LIN {X 0,Y 468.037,Z 394.262,A -85,B 0,C 180,E1 -7685.847,E2 -7685.847} C_VEL
LIN {X 0,Y 468.13,Z 390.567,A -85,B 0,C 180,E1 -7687.99,E2 -7687.99} C_VEL
LIN {X 0,Y 467.913,Z 386.87,A -85,B 0,C 180,E1 -7690.23,E2 -7690.23} C_VEL
LIN {X 0,Y 467.598,Z 384.87,A -85,B 0,C 180,E1 -7691.544,E2 -7691.544} C_VEL
LIN {X 0,Y 467.567,Z 384.871,A -85,B 0,C 180,E1 -7695.053,E2 -7695.053} C_VEL
LIN {X 0,Y 467.59,Z 384.868,A -85,B 0,C 180,E1 -7697.44,E2 -7697.44} C_VEL
LIN {X 0,Y 467.62,Z 384.864,A -85,B 0,C 180,E1 -7700.859,E2 -7700.859} C_VEL
LIN {X 0,Y 467.565,Z 384.872,A -85,B 0,C 180,E1 -7704.26,E2 -7704.26} C_VEL
LIN {X 0,Y 467.583,Z 384.868,A -85,B 0,C 180,E1 -7707.321,E2 -7707.321} C_VEL
LIN {X 0,Y 467.572,Z 384.871,A -85,B 0,C 180,E1 -7710.667,E2 -7710.667} C_VEL
LIN {X 0,Y 467.614,Z 384.861,A -85,B 0,C 180,E1 -7713.2,E2 -7713.2} C_VEL
LIN {X 0,Y 467.591,Z 384.863,A -85,B 0,C 180,E1 -7716.469,E2 -7716.469} C_VEL
LIN {X 0,Y 467.626,Z 384.859,A -85,B 0,C 180,E1 -7719.777,E2 -7719.777} C_VEL
LIN {X 0,Y 467.611,Z 384.862,A -85,B 0,C 180,E1 -7722.507,E2 -7722.507} C_VEL
LIN {X 0,Y 467.612,Z 384.864,A -85,B 0,C 180,E1 -7725.197,E2 -7725.197} C_VEL
LIN {X 0,Y 467.658,Z 384.855,A -85,B 0,C 180,E1 -7727.855,E2 -7727.855} C_VEL
LIN {X 0,Y 467.683,Z 384.852,A -85,B 0,C 180,E1 -7731.357,E2 -7731.357} C_VEL
LIN {X 0,Y 467.745,Z 384.845,A -85,B 0,C 180,E1 -7733.963,E2 -7733.963} C_VEL
LIN {X 0,Y 467.862,Z 384.83,A -85,B 0,C 180,E1 -7737.417,E2 -7737.417} C_VEL
LIN {X 0,Y 467.885,Z 384.831,A -85,B 0,C 180,E1 -7740,E2 -7740} C_VEL
LIN {X 0,Y 467.861,Z 384.829,A -85,B 0,C 180,E1 -7742.583,E2 -7742.583} C_VEL
LIN {X 0,Y 467.746,Z 384.845,A -85,B 0,C 180,E1 -7746.037,E2 -7746.037} C_VEL
LIN {X 0,Y 467.683,Z 384.852,A -85,B 0,C 180,E1 -7748.643,E2 -7748.643} C_VEL
LIN {X 0,Y 467.658,Z 384.855,A -85,B 0,C 180,E1 -7752.145,E2 -7752.145} C_VEL
LIN {X 0,Y 467.658,Z 384.856,A -85,B 0,C 180,E1 -7755.694,E2 -7755.694} C_VEL
LIN {X 0,Y 467.62,Z 384.86,A -85,B 0,C 180,E1 -7758.765,E2 -7758.765} C_VEL
LIN {X 0,Y 467.583,Z 384.868,A -85,B 0,C 180,E1 -7761.269,E2 -7761.269} C_VEL
LIN {X 0,Y 467.576,Z 384.867,A -85,B 0,C 180,E1 -7763.943,E2 -7763.943} C_VEL
LIN {X 0,Y 467.618,Z 384.86,A -85,B 0,C 180,E1 -7766.8,E2 -7766.8} C_VEL
LIN {X 0,Y 467.556,Z 384.868,A -85,B 0,C 180,E1 -7769.738,E2 -7769.738} C_VEL
LIN {X 0,Y 467.585,Z 384.867,A -85,B 0,C 180,E1 -7772.758,E2 -7772.758} C_VEL
LIN {X 0,Y 467.559,Z 384.871,A -85,B 0,C 180,E1 -7775.889,E2 -7775.889} C_VEL
LIN {X 0,Y 467.585,Z 384.867,A -85,B 0,C 180,E1 -7779.145,E2 -7779.145} C_VEL
LIN {X 0,Y 467.588,Z 384.866,A -85,B 0,C 180,E1 -7782.567,E2 -7782.567} C_VEL
LIN {X 0,Y 467.572,Z 384.869,A -85,B 0,C 180,E1 -7785.053,E2 -7785.053} C_VEL
LIN {X 0,Y 467.59,Z 384.867,A -85,B 0,C 180,E1 -7787.44,E2 -7787.44} C_VEL
LIN {X 0,Y 467.569,Z 384.87,A -85,B 0,C 180,E1 -7789.735,E2 -7789.735} C_VEL
LIN {X 0,Y 467.756,Z 387.867,A -85,B 0,C 180,E1 -7791.974,E2 -7791.974} C_VEL
LIN {X 0,Y 467.68,Z 392.609,A -85,B 0,C 180,E1 -7795.177,E2 -7795.177} C_VEL
LIN {X 0,Y 467.509,Z 397.368,A -85,B 0,C 180,E1 -7798.254,E2 -7798.254} C_VEL
LIN {X 0,Y 467.314,Z 402.123,A -85,B 0,C 180,E1 -7801.233,E2 -7801.233} C_VEL
LIN {X 0,Y 467.189,Z 407.463,A -85,B 0,C 180,E1 -7804.501,E2 -7804.501} C_VEL
LIN {X 0,Y 467.08,Z 411.589,A -85,B 0,C 180,E1 -7806.97,E2 -7806.97} C_VEL
LIN {X 0,Y 466.947,Z 416.313,A -85,B 0,C 180,E1 -7809.747,E2 -7809.747} C_VEL
LIN {X 0,Y 466.908,Z 419.366,A -85,B 0,C 180,E1 -7811.43,E2 -7811.43} C_VEL
LIN {X 0,Y 470.476,Z 434.191,A -85,B 0,C 180,E1 -7811.94,E2 -7811.94} C_VEL
LIN {X 0,Y 471.792,Z 441.602,A -85,B 0,C 180,E1 -7812.248,E2 -7812.248} C_VEL
LIN {X 0,Y 471.556,Z 447.954,A -85,B 0,C 180,E1 -7812.5,E2 -7812.5} C_VEL
LIN {X 0,Y 470.818,Z 453.507,A -85,B 0,C 180,E1 -7812.727,E2 -7812.727} C_VEL
LIN {X 0,Y 467.754,Z 462.443,A -85,B 0,C 180,E1 -7813.094,E2 -7813.094} C_VEL
LIN {X 0,Y 464.513,Z 471.086,A -85,B 0,C 180,E1 -7813.54,E2 -7813.54} C_VEL
LIN {X 0,Y 463.507,Z 476.182,A -85,B 0,C 180,E1 -7813.888,E2 -7813.888} C_VEL
LIN {X 0,Y 462.736,Z 487.332,A -85,B 0,C 180,E1 -7814.812,E2 -7814.812} C_VEL
LIN {X 0,Y 462.061,Z 498.248,A -85,B 0,C 180,E1 -7815.915,E2 -7815.915} C_VEL
LIN {X 0,Y 461.458,Z 507.914,A -85,B 0,C 180,E1 -7817.09,E2 -7817.09} C_VEL
LIN {X 0,Y 461.01,Z 516.552,A -85,B 0,C 180,E1 -7818.347,E2 -7818.347} C_VEL
LIN {X 0,Y 460.484,Z 524.187,A -85,B 0,C 180,E1 -7819.669,E2 -7819.669} C_VEL
LIN {X 0,Y 460.097,Z 531.463,A -85,B 0,C 180,E1 -7821.214,E2 -7821.214} C_VEL
LIN {X 0,Y 459.838,Z 537.999,A -85,B 0,C 180,E1 -7822.977,E2 -7822.977} C_VEL
LIN {X 0,Y 459.713,Z 542.902,A -85,B 0,C 180,E1 -7824.737,E2 -7824.737} C_VEL
LIN {X 0,Y 459.585,Z 546.316,A -85,B 0,C 180,E1 -7826.493,E2 -7826.493} C_VEL
LIN {X 0,Y 459.519,Z 548.346,A -85,B 0,C 180,E1 -7828.247,E2 -7828.247} C_VEL
LIN {X 0,Y 459.5,Z 549.045,A -85,B 0,C 180,E1 -7830,E2 -7830} C_VEL
LIN {X 0,Y 459.518,Z 548.421,A -85,B 0,C 180,E1 -7831.753,E2 -7831.753} C_VEL
LIN {X 0,Y 459.585,Z 546.46,A -85,B 0,C 180,E1 -7833.507,E2 -7833.507} C_VEL
LIN {X 0,Y 459.707,Z 543.116,A -85,B 0,C 180,E1 -7835.263,E2 -7835.263} C_VEL
LIN {X 0,Y 459.794,Z 538.292,A -85,B 0,C 180,E1 -7837.024,E2 -7837.024} C_VEL
LIN {X 0,Y 460.086,Z 531.831,A -85,B 0,C 180,E1 -7838.787,E2 -7838.787} C_VEL
LIN {X 0,Y 460.443,Z 524.638,A -85,B 0,C 180,E1 -7840.332,E2 -7840.332} C_VEL
LIN {X 0,Y 461.045,Z 515.741,A -85,B 0,C 180,E1 -7841.876,E2 -7841.876} C_VEL
LIN {X 0,Y 461.588,Z 506.395,A -85,B 0,C 180,E1 -7843.202,E2 -7843.202} C_VEL
LIN {X 0,Y 462.235,Z 496.043,A -85,B 0,C 180,E1 -7844.417,E2 -7844.417} C_VEL
LIN {X 0,Y 462.959,Z 484.619,A -85,B 0,C 180,E1 -7845.519,E2 -7845.519} C_VEL
LIN {X 0,Y 463.727,Z 471.957,A -85,B 0,C 180,E1 -7846.509,E2 -7846.509} C_VEL
LIN {X 0,Y 464.367,Z 459.383,A -85,B 0,C 180,E1 -7847.294,E2 -7847.294} C_VEL
LIN {X 0,Y 464.879,Z 446.27,A -85,B 0,C 180,E1 -7847.929,E2 -7847.929} C_VEL
LIN {X 0,Y 464.878,Z 441.114,A -85,B 0,C 180,E1 -7848.138,E2 -7848.138} C_VEL
LIN {X 0,Y 461.867,Z 427.454,A -85,B 0,C 180,E1 -7848.697,E2 -7848.697} C_VEL
LIN {X 0,Y 459.864,Z 419.255,A -85,B 0,C 180,E1 -7848.975,E2 -7848.975} C_VEL
LIN {X 0,Y 459.964,Z 413.379,A -85,B 0,C 180,E1 -7852.457,E2 -7852.457} C_VEL
LIN {X 0,Y 460.119,Z 408.047,A -85,B 0,C 180,E1 -7855.685,E2 -7855.685} C_VEL
LIN {X 0,Y 460.223,Z 403.902,A -85,B 0,C 180,E1 -7858.255,E2 -7858.255} C_VEL
LIN {X 0,Y 460.45,Z 399.139,A -85,B 0,C 180,E1 -7861.268,E2 -7861.268} C_VEL
LIN {X 0,Y 460.615,Z 394.161,A -85,B 0,C 180,E1 -7864.52,E2 -7864.52} C_VEL
LIN {X 0,Y 460.755,Z 389.63,A -85,B 0,C 180,E1 -7867.599,E2 -7867.599} C_VEL
LIN {X 0,Y 460.574,Z 385.879,A -85,B 0,C 180,E1 -7870.274,E2 -7870.274} C_VEL
LIN {X 0,Y 460.512,Z 385.75,A -85,B 0,C 180,E1 -7873.374,E2 -7873.374} C_VEL
LIN {X 0,Y 460.503,Z 385.751,A -85,B 0,C 180,E1 -7876.625,E2 -7876.625} C_VEL
LIN {X 0,Y 460.544,Z 385.745,A -85,B 0,C 180,E1 -7879.731,E2 -7879.731} C_VEL
LIN {X 0,Y 460.53,Z 385.746,A -85,B 0,C 180,E1 -7882.519,E2 -7882.519} C_VEL
LIN {X 0,Y 460.552,Z 385.742,A -85,B 0,C 180,E1 -7885.624,E2 -7885.624} C_VEL
LIN {X 0,Y 460.54,Z 385.742,A -85,B 0,C 180,E1 -7888.745,E2 -7888.745} C_VEL
LIN {X 0,Y 460.592,Z 385.738,A -85,B 0,C 180,E1 -7892.252,E2 -7892.252} C_VEL
LIN {X 0,Y 460.562,Z 385.74,A -85,B 0,C 180,E1 -7894.705,E2 -7894.705} C_VEL
LIN {X 0,Y 460.514,Z 385.748,A -85,B 0,C 180,E1 -7897.571,E2 -7897.571} C_VEL
LIN {X 0,Y 460.572,Z 385.738,A -85,B 0,C 180,E1 -7900.385,E2 -7900.385} C_VEL
LIN {X 0,Y 460.567,Z 385.738,A -85,B 0,C 180,E1 -7903.146,E2 -7903.146} C_VEL
LIN {X 0,Y 460.561,Z 385.74,A -85,B 0,C 180,E1 -7905.868,E2 -7905.868} C_VEL
LIN {X 0,Y 460.614,Z 385.737,A -85,B 0,C 180,E1 -7908.559,E2 -7908.559} C_VEL
LIN {X 0,Y 460.698,Z 385.725,A -85,B 0,C 180,E1 -7912.109,E2 -7912.109} C_VEL
LIN {X 0,Y 460.7,Z 385.723,A -85,B 0,C 180,E1 -7914.748,E2 -7914.748} C_VEL
LIN {X 0,Y 460.803,Z 385.709,A -85,B 0,C 180,E1 -7917.377,E2 -7917.377} C_VEL
LIN {X 0,Y 460.856,Z 385.708,A -85,B 0,C 180,E1 -7920,E2 -7920} C_VEL
LIN {X 0,Y 460.828,Z 385.706,A -85,B 0,C 180,E1 -7922.622,E2 -7922.622} C_VEL
LIN {X 0,Y 460.713,Z 385.721,A -85,B 0,C 180,E1 -7926.13,E2 -7926.13} C_VEL
LIN {X 0,Y 460.631,Z 385.731,A -85,B 0,C 180,E1 -7928.776,E2 -7928.776} C_VEL
LIN {X 0,Y 460.616,Z 385.733,A -85,B 0,C 180,E1 -7932.445,E2 -7932.445} C_VEL
LIN {X 0,Y 460.603,Z 385.737,A -85,B 0,C 180,E1 -7935.997,E2 -7935.997} C_VEL
LIN {X 0,Y 460.574,Z 385.738,A -85,B 0,C 180,E1 -7938.902,E2 -7938.902} C_VEL
LIN {X 0,Y 460.519,Z 385.746,A -85,B 0,C 180,E1 -7941.485,E2 -7941.485} C_VEL
LIN {X 0,Y 460.545,Z 385.743,A -85,B 0,C 180,E1 -7944.332,E2 -7944.332} C_VEL
LIN {X 0,Y 460.582,Z 385.737,A -85,B 0,C 180,E1 -7947.243,E2 -7947.243} C_VEL
LIN {X 0,Y 460.513,Z 385.744,A -85,B 0,C 180,E1 -7950.24,E2 -7950.24} C_VEL
LIN {X 0,Y 460.532,Z 385.744,A -85,B 0,C 180,E1 -7953.325,E2 -7953.325} C_VEL
LIN {X 0,Y 460.482,Z 385.751,A -85,B 0,C 180,E1 -7956.529,E2 -7956.529} C_VEL
LIN {X 0,Y 460.58,Z 385.739,A -85,B 0,C 180,E1 -7959.857,E2 -7959.857} C_VEL
LIN {X 0,Y 460.514,Z 385.747,A -85,B 0,C 180,E1 -7962.9,E2 -7962.9} C_VEL
LIN {X 0,Y 460.511,Z 385.75,A -85,B 0,C 180,E1 -7965.831,E2 -7965.831} C_VEL
LIN {X 0,Y 460.578,Z 385.905,A -85,B 0,C 180,E1 -7968.391,E2 -7968.391} C_VEL
LIN {X 0,Y 461.077,Z 390.044,A -85,B 0,C 180,E1 -7971.021,E2 -7971.021} C_VEL
LIN {X 0,Y 461.049,Z 394.238,A -85,B 0,C 180,E1 -7973.523,E2 -7973.523} C_VEL
LIN {X 0,Y 460.771,Z 399.769,A -85,B 0,C 180,E1 -7976.695,E2 -7976.695} C_VEL
LIN {X 0,Y 460.523,Z 405.31,A -85,B 0,C 180,E1 -7979.761,E2 -7979.761} C_VEL
LIN {X 0,Y 460.344,Z 410.858,A -85,B 0,C 180,E1 -7982.741,E2 -7982.741} C_VEL
LIN {X 0,Y 460.14,Z 416.417,A -85,B 0,C 180,E1 -7985.645,E2 -7985.645} C_VEL
LIN {X 0,Y 460.006,Z 422.481,A -85,B 0,C 180,E1 -7988.743,E2 -7988.743} C_VEL
LIN {X 0,Y 459.895,Z 427.136,A -85,B 0,C 180,E1 -7991.074,E2 -7991.074} C_VEL
LIN {X 0,Y 463.203,Z 441.778,A -85,B 0,C 180,E1 -7991.567,E2 -7991.567} C_VEL
LIN {X 0,Y 464.921,Z 450.797,A -85,B 0,C 180,E1 -7991.95,E2 -7991.95} C_VEL
LIN {X 0,Y 464.492,Z 463.02,A -85,B 0,C 180,E1 -7992.486,E2 -7992.486} C_VEL
LIN {X 0,Y 463.786,Z 476.719,A -85,B 0,C 180,E1 -7993.267,E2 -7993.267} C_VEL
LIN {X 0,Y 463.109,Z 488.85,A -85,B 0,C 180,E1 -7994.147,E2 -7994.147} C_VEL
LIN {X 0,Y 462.43,Z 499.993,A -85,B 0,C 180,E1 -7995.139,E2 -7995.139} C_VEL
LIN {X 0,Y 461.69,Z 511.188,A -85,B 0,C 180,E1 -7996.352,E2 -7996.352} C_VEL
LIN {X 0,Y 461.077,Z 521.227,A -85,B 0,C 180,E1 -7997.678,E2 -7997.678} C_VEL
LIN {X 0,Y 460.622,Z 529.565,A -85,B 0,C 180,E1 -7999.005,E2 -7999.005} C_VEL
LIN {X 0,Y 460.167,Z 537.534,A -85,B 0,C 180,E1 -8000.55,E2 -8000.55} C_VEL
LIN {X 0,Y 459.848,Z 543.951,A -85,B 0,C 180,E1 -8002.094,E2 -8002.094} C_VEL
LIN {X 0,Y 459.697,Z 549.639,A -85,B 0,C 180,E1 -8003.856,E2 -8003.856} C_VEL
LIN {X 0,Y 459.676,Z 551.888,A -85,B 0,C 180,E1 -8004.737,E2 -8004.737} C_VEL
LIN {X 0,Y 459.548,Z 555.286,A -85,B 0,C 180,E1 -8006.493,E2 -8006.493} C_VEL
LIN {X 0,Y 459.514,Z 557.296,A -85,B 0,C 180,E1 -8008.247,E2 -8008.247} C_VEL
LIN {X 0,Y 459.499,Z 557.962,A -85,B 0,C 180,E1 -8010,E2 -8010} C_VEL
LIN {X 0,Y 459.514,Z 557.297,A -85,B 0,C 180,E1 -8011.753,E2 -8011.753} C_VEL
LIN {X 0,Y 459.548,Z 555.29,A -85,B 0,C 180,E1 -8013.507,E2 -8013.507} C_VEL
LIN {X 0,Y 459.675,Z 551.891,A -85,B 0,C 180,E1 -8015.263,E2 -8015.263} C_VEL
LIN {X 0,Y 459.739,Z 546.998,A -85,B 0,C 180,E1 -8017.025,E2 -8017.025} C_VEL
LIN {X 0,Y 460.042,Z 540.468,A -85,B 0,C 180,E1 -8018.787,E2 -8018.787} C_VEL
LIN {X 0,Y 460.37,Z 533.2,A -85,B 0,C 180,E1 -8020.333,E2 -8020.333} C_VEL
LIN {X 0,Y 460.98,Z 524.2,A -85,B 0,C 180,E1 -8021.877,E2 -8021.877} C_VEL
LIN {X 0,Y 461.502,Z 514.753,A -85,B 0,C 180,E1 -8023.204,E2 -8023.204} C_VEL
LIN {X 0,Y 462.124,Z 504.293,A -85,B 0,C 180,E1 -8024.42,E2 -8024.42} C_VEL
LIN {X 0,Y 462.87,Z 492.752,A -85,B 0,C 180,E1 -8025.522,E2 -8025.522} C_VEL
LIN {X 0,Y 463.62,Z 479.947,A -85,B 0,C 180,E1 -8026.513,E2 -8026.513} C_VEL
LIN {X 0,Y 464.325,Z 466.553,A -85,B 0,C 180,E1 -8027.331,E2 -8027.331} C_VEL
LIN {X 0,Y 464.838,Z 453.547,A -85,B 0,C 180,E1 -8027.941,E2 -8027.941} C_VEL
LIN {X 0,Y 464.782,Z 449.968,A -85,B 0,C 180,E1 -8028.085,E2 -8028.085} C_VEL
LIN {X 0,Y 461.942,Z 435.895,A -85,B 0,C 180,E1 -8028.648,E2 -8028.648} C_VEL
LIN {X 0,Y 459.916,Z 427.098,A -85,B 0,C 180,E1 -8028.94,E2 -8028.94} C_VEL
LIN {X 0,Y 460.047,Z 420.117,A -85,B 0,C 180,E1 -8032.452,E2 -8032.452} C_VEL
LIN {X 0,Y 460.23,Z 413.791,A -85,B 0,C 180,E1 -8035.714,E2 -8035.714} C_VEL
LIN {X 0,Y 460.374,Z 408.996,A -85,B 0,C 180,E1 -8038.245,E2 -8038.245} C_VEL
LIN {X 0,Y 460.633,Z 403.347,A -85,B 0,C 180,E1 -8041.306,E2 -8041.306} C_VEL
LIN {X 0,Y 460.892,Z 397.528,A -85,B 0,C 180,E1 -8044.57,E2 -8044.57} C_VEL
LIN {X 0,Y 461.125,Z 392.357,A -85,B 0,C 180,E1 -8047.577,E2 -8047.577} C_VEL
LIN {X 0,Y 460.973,Z 388.68,A -85,B 0,C 180,E1 -8049.817,E2 -8049.817} C_VEL
LIN {X 0,Y 460.57,Z 385.745,A -85,B 0,C 180,E1 -8051.733,E2 -8051.733} C_VEL
LIN {X 0,Y 460.514,Z 385.748,A -85,B 0,C 180,E1 -8055.411,E2 -8055.411} C_VEL
LIN {X 0,Y 460.536,Z 385.745,A -85,B 0,C 180,E1 -8058.397,E2 -8058.397} C_VEL
LIN {X 0,Y 460.549,Z 385.745,A -85,B 0,C 180,E1 -8061.269,E2 -8061.269} C_VEL
LIN {X 0,Y 460.515,Z 385.749,A -85,B 0,C 180,E1 -8064.555,E2 -8064.555} C_VEL
LIN {X 0,Y 460.533,Z 385.747,A -85,B 0,C 180,E1 -8067.716,E2 -8067.716} C_VEL
LIN {X 0,Y 460.541,Z 385.747,A -85,B 0,C 180,E1 -8070.769,E2 -8070.769} C_VEL
LIN {X 0,Y 460.557,Z 385.742,A -85,B 0,C 180,E1 -8073.734,E2 -8073.734} C_VEL
LIN {X 0,Y 460.545,Z 385.741,A -85,B 0,C 180,E1 -8076.624,E2 -8076.624} C_VEL
LIN {X 0,Y 460.554,Z 385.741,A -85,B 0,C 180,E1 -8079.453,E2 -8079.453} C_VEL
LIN {X 0,Y 460.561,Z 385.742,A -85,B 0,C 180,E1 -8082.23,E2 -8082.23} C_VEL
LIN {X 0,Y 460.574,Z 385.738,A -85,B 0,C 180,E1 -8084.965,E2 -8084.965} C_VEL
LIN {X 0,Y 460.613,Z 385.736,A -85,B 0,C 180,E1 -8088.559,E2 -8088.559} C_VEL
LIN {X 0,Y 460.697,Z 385.723,A -85,B 0,C 180,E1 -8092.109,E2 -8092.109} C_VEL
LIN {X 0,Y 460.699,Z 385.723,A -85,B 0,C 180,E1 -8094.748,E2 -8094.748} C_VEL
LIN {X 0,Y 460.827,Z 385.706,A -85,B 0,C 180,E1 -8097.378,E2 -8097.378} C_VEL
LIN {X 0,Y 460.856,Z 385.707,A -85,B 0,C 180,E1 -8100,E2 -8100} C_VEL
LIN {X 0,Y 460.802,Z 385.709,A -85,B 0,C 180,E1 -8102.623,E2 -8102.623} C_VEL
LIN {X 0,Y 460.712,Z 385.722,A -85,B 0,C 180,E1 -8106.13,E2 -8106.13} C_VEL
LIN {X 0,Y 460.63,Z 385.73,A -85,B 0,C 180,E1 -8108.776,E2 -8108.776} C_VEL
LIN {X 0,Y 460.615,Z 385.733,A -85,B 0,C 180,E1 -8112.445,E2 -8112.445} C_VEL
LIN {X 0,Y 460.624,Z 385.734,A -85,B 0,C 180,E1 -8116.007,E2 -8116.007} C_VEL
LIN {X 0,Y 460.572,Z 385.742,A -85,B 0,C 180,E1 -8119.615,E2 -8119.615} C_VEL
LIN {X 0,Y 460.514,Z 385.747,A -85,B 0,C 180,E1 -8122.429,E2 -8122.429} C_VEL
LIN {X 0,Y 460.57,Z 385.742,A -85,B 0,C 180,E1 -8125.802,E2 -8125.802} C_VEL
LIN {X 0,Y 460.557,Z 385.74,A -85,B 0,C 180,E1 -8128.233,E2 -8128.233} C_VEL
LIN {X 0,Y 460.522,Z 385.745,A -85,B 0,C 180,E1 -8131.283,E2 -8131.283} C_VEL
LIN {X 0,Y 460.536,Z 385.744,A -85,B 0,C 180,E1 -8134.506,E2 -8134.506} C_VEL
LIN {X 0,Y 460.531,Z 385.745,A -85,B 0,C 180,E1 -8137.62,E2 -8137.62} C_VEL
LIN {X 0,Y 460.544,Z 385.744,A -85,B 0,C 180,E1 -8140.27,E2 -8140.27} C_VEL
LIN {X 0,Y 460.501,Z 385.749,A -85,B 0,C 180,E1 -8143.375,E2 -8143.375} C_VEL
LIN {X 0,Y 460.515,Z 385.748,A -85,B 0,C 180,E1 -8146.626,E2 -8146.626} C_VEL
LIN {X 0,Y 460.537,Z 385.75,A -85,B 0,C 180,E1 -8149.732,E2 -8149.732} C_VEL
LIN {X 0,Y 460.756,Z 389.603,A -85,B 0,C 180,E1 -8152.483,E2 -8152.483} C_VEL
LIN {X 0,Y 460.65,Z 394.238,A -85,B 0,C 180,E1 -8155.633,E2 -8155.633} C_VEL
LIN {X 0,Y 460.446,Z 399,A -85,B 0,C 180,E1 -8158.738,E2 -8158.738} C_VEL
LIN {X 0,Y 460.223,Z 403.751,A -85,B 0,C 180,E1 -8161.745,E2 -8161.745} C_VEL
LIN {X 0,Y 460.122,Z 408.492,A -85,B 0,C 180,E1 -8164.68,E2 -8164.68} C_VEL
LIN {X 0,Y 459.975,Z 413.225,A -85,B 0,C 180,E1 -8167.544,E2 -8167.544} C_VEL
LIN {X 0,Y 459.85,Z 417.954,A -85,B 0,C 180,E1 -8170.353,E2 -8170.353} C_VEL
LIN {X 0,Y 459.862,Z 419.338,A -85,B 0,C 180,E1 -8171.132,E2 -8171.132} C_VEL
LIN {X 0,Y 463.348,Z 433.67,A -85,B 0,C 180,E1 -8171.633,E2 -8171.633} C_VEL
LIN {X 0,Y 465.03,Z 442.126,A -85,B 0,C 180,E1 -8171.997,E2 -8171.997} C_VEL
LIN {X 0,Y 464.506,Z 455.87,A -85,B 0,C 180,E1 -8172.606,E2 -8172.606} C_VEL
LIN {X 0,Y 463.869,Z 469.112,A -85,B 0,C 180,E1 -8173.383,E2 -8173.383} C_VEL
LIN {X 0,Y 463.507,Z 476.182,A -85,B 0,C 180,E1 -8173.888,E2 -8173.888} C_VEL
LIN {X 0,Y 462.509,Z 481.258,A -85,B 0,C 180,E1 -8174.261,E2 -8174.261} C_VEL
LIN {X 0,Y 459.2,Z 489.238,A -85,B 0,C 180,E1 -8174.873,E2 -8174.873} C_VEL
LIN {X 0,Y 455.935,Z 496.805,A -85,B 0,C 180,E1 -8175.547,E2 -8175.547} C_VEL
LIN {X 0,Y 454.968,Z 501.163,A -85,B 0,C 180,E1 -8176.025,E2 -8176.025} C_VEL
LIN {X 0,Y 454.322,Z 510.322,A -85,B 0,C 180,E1 -8177.211,E2 -8177.211} C_VEL
LIN {X 0,Y 453.829,Z 519.326,A -85,B 0,C 180,E1 -8178.612,E2 -8178.612} C_VEL
LIN {X 0,Y 453.316,Z 527.585,A -85,B 0,C 180,E1 -8180.181,E2 -8180.181} C_VEL
LIN {X 0,Y 452.968,Z 533.338,A -85,B 0,C 180,E1 -8181.524,E2 -8181.524} C_VEL
LIN {X 0,Y 452.752,Z 538.07,A -85,B 0,C 180,E1 -8182.867,E2 -8182.867} C_VEL
LIN {X 0,Y 452.629,Z 542.972,A -85,B 0,C 180,E1 -8184.655,E2 -8184.655} C_VEL
LIN {X 0,Y 452.484,Z 546.386,A -85,B 0,C 180,E1 -8186.438,E2 -8186.438} C_VEL
LIN {X 0,Y 452.435,Z 548.415,A -85,B 0,C 180,E1 -8188.22,E2 -8188.22} C_VEL
LIN {X 0,Y 452.406,Z 549.114,A -85,B 0,C 180,E1 -8190,E2 -8190} C_VEL
LIN {X 0,Y 452.435,Z 548.49,A -85,B 0,C 180,E1 -8191.78,E2 -8191.78} C_VEL
LIN {X 0,Y 452.483,Z 546.529,A -85,B 0,C 180,E1 -8193.562,E2 -8193.562} C_VEL
LIN {X 0,Y 452.621,Z 543.184,A -85,B 0,C 180,E1 -8195.346,E2 -8195.346} C_VEL
LIN {X 0,Y 452.729,Z 538.359,A -85,B 0,C 180,E1 -8197.134,E2 -8197.134} C_VEL
LIN {X 0,Y 453.055,Z 531.898,A -85,B 0,C 180,E1 -8198.924,E2 -8198.924} C_VEL
LIN {X 0,Y 453.406,Z 524.705,A -85,B 0,C 180,E1 -8200.494,E2 -8200.494} C_VEL
LIN {X 0,Y 453.972,Z 517.167,A -85,B 0,C 180,E1 -8201.837,E2 -8201.837} C_VEL
LIN {X 0,Y 454.525,Z 507.883,A -85,B 0,C 180,E1 -8203.216,E2 -8203.216} C_VEL
LIN {X 0,Y 455.27,Z 497.15,A -85,B 0,C 180,E1 -8204.528,E2 -8204.528} C_VEL
LIN {X 0,Y 456.044,Z 485.97,A -85,B 0,C 180,E1 -8205.646,E2 -8205.646} C_VEL
LIN {X 0,Y 456.826,Z 473.599,A -85,B 0,C 180,E1 -8206.651,E2 -8206.651} C_VEL
LIN {X 0,Y 457.474,Z 461.618,A -85,B 0,C 180,E1 -8207.436,E2 -8207.436} C_VEL
LIN {X 0,Y 458.029,Z 448.537,A -85,B 0,C 180,E1 -8208.108,E2 -8208.108} C_VEL
LIN {X 0,Y 458.146,Z 442.462,A -85,B 0,C 180,E1 -8208.365,E2 -8208.365} C_VEL
LIN {X 0,Y 455.135,Z 428.794,A -85,B 0,C 180,E1 -8208.951,E2 -8208.951} C_VEL
LIN {X 0,Y 452.775,Z 419.323,A -85,B 0,C 180,E1 -8209.283,E2 -8209.283} C_VEL
LIN {X 0,Y 452.853,Z 415.019,A -85,B 0,C 180,E1 -8211.868,E2 -8211.868} C_VEL
LIN {X 0,Y 453.008,Z 410.279,A -85,B 0,C 180,E1 -8214.764,E2 -8214.764} C_VEL
LIN {X 0,Y 453.143,Z 405.321,A -85,B 0,C 180,E1 -8217.866,E2 -8217.866} C_VEL
LIN {X 0,Y 453.345,Z 400.775,A -85,B 0,C 180,E1 -8220.77,E2 -8220.77} C_VEL
LIN {X 0,Y 453.539,Z 396.016,A -85,B 0,C 180,E1 -8223.908,E2 -8223.908} C_VEL
LIN {X 0,Y 453.711,Z 391.246,A -85,B 0,C 180,E1 -8227.165,E2 -8227.165} C_VEL
LIN {X 0,Y 453.632,Z 388.074,A -85,B 0,C 180,E1 -8229.435,E2 -8229.435} C_VEL
LIN {X 0,Y 453.519,Z 386.623,A -85,B 0,C 180,E1 -8230.606,E2 -8230.606} C_VEL
LIN {X 0,Y 453.476,Z 386.626,A -85,B 0,C 180,E1 -8234.22,E2 -8234.22} C_VEL
LIN {X 0,Y 453.466,Z 386.626,A -85,B 0,C 180,E1 -8237.005,E2 -8237.005} C_VEL
LIN {X 0,Y 453.497,Z 386.624,A -85,B 0,C 180,E1 -8239.409,E2 -8239.409} C_VEL
LIN {X 0,Y 453.476,Z 386.622,A -85,B 0,C 180,E1 -8242.223,E2 -8242.223} C_VEL
LIN {X 0,Y 453.492,Z 386.62,A -85,B 0,C 180,E1 -8245.222,E2 -8245.222} C_VEL
LIN {X 0,Y 453.469,Z 386.622,A -85,B 0,C 180,E1 -8248.475,E2 -8248.475} C_VEL
LIN {X 0,Y 453.54,Z 386.615,A -85,B 0,C 180,E1 -8252.039,E2 -8252.039} C_VEL
LIN {X 0,Y 453.517,Z 386.618,A -85,B 0,C 180,E1 -8255.266,E2 -8255.266} C_VEL
LIN {X 0,Y 453.483,Z 386.621,A -85,B 0,C 180,E1 -8258.415,E2 -8258.415} C_VEL
LIN {X 0,Y 453.525,Z 386.617,A -85,B 0,C 180,E1 -8261.009,E2 -8261.009} C_VEL
LIN {X 0,Y 453.572,Z 386.614,A -85,B 0,C 180,E1 -8263.88,E2 -8263.88} C_VEL
LIN {X 0,Y 453.567,Z 386.612,A -85,B 0,C 180,E1 -8267.471,E2 -8267.471} C_VEL
LIN {X 0,Y 453.595,Z 386.606,A -85,B 0,C 180,E1 -8271.087,E2 -8271.087} C_VEL
LIN {X 0,Y 453.681,Z 386.599,A -85,B 0,C 180,E1 -8273.775,E2 -8273.775} C_VEL
LIN {X 0,Y 453.747,Z 386.588,A -85,B 0,C 180,E1 -8277.337,E2 -8277.337} C_VEL
LIN {X 0,Y 453.826,Z 386.583,A -85,B 0,C 180,E1 -8280,E2 -8280} C_VEL
LIN {X 0,Y 453.768,Z 386.586,A -85,B 0,C 180,E1 -8282.663,E2 -8282.663} C_VEL
LIN {X 0,Y 453.68,Z 386.597,A -85,B 0,C 180,E1 -8286.225,E2 -8286.225} C_VEL
LIN {X 0,Y 453.595,Z 386.607,A -85,B 0,C 180,E1 -8288.913,E2 -8288.913} C_VEL
LIN {X 0,Y 453.566,Z 386.611,A -85,B 0,C 180,E1 -8292.529,E2 -8292.529} C_VEL
LIN {X 0,Y 453.548,Z 386.618,A -85,B 0,C 180,E1 -8296.196,E2 -8296.196} C_VEL
LIN {X 0,Y 453.524,Z 386.617,A -85,B 0,C 180,E1 -8299.041,E2 -8299.041} C_VEL
LIN {X 0,Y 453.479,Z 386.621,A -85,B 0,C 180,E1 -8301.836,E2 -8301.836} C_VEL
LIN {X 0,Y 453.517,Z 386.618,A -85,B 0,C 180,E1 -8304.734,E2 -8304.734} C_VEL
LIN {X 0,Y 453.54,Z 386.615,A -85,B 0,C 180,E1 -8307.961,E2 -8307.961} C_VEL
LIN {X 0,Y 453.468,Z 386.623,A -85,B 0,C 180,E1 -8311.525,E2 -8311.525} C_VEL
LIN {X 0,Y 453.492,Z 386.621,A -85,B 0,C 180,E1 -8314.778,E2 -8314.778} C_VEL
LIN {X 0,Y 453.488,Z 386.623,A -85,B 0,C 180,E1 -8318.309,E2 -8318.309} C_VEL
LIN {X 0,Y 453.518,Z 386.623,A -85,B 0,C 180,E1 -8320.606,E2 -8320.606} C_VEL
LIN {X 0,Y 453.465,Z 386.626,A -85,B 0,C 180,E1 -8324.221,E2 -8324.221} C_VEL
LIN {X 0,Y 453.465,Z 386.63,A -85,B 0,C 180,E1 -8327.005,E2 -8327.005} C_VEL
LIN {X 0,Y 453.54,Z 386.827,A -85,B 0,C 180,E1 -8328.216,E2 -8328.216} C_VEL
LIN {X 0,Y 454.031,Z 390.68,A -85,B 0,C 180,E1 -8330.711,E2 -8330.711} C_VEL
LIN {X 0,Y 454.059,Z 394.202,A -85,B 0,C 180,E1 -8332.868,E2 -8332.868} C_VEL
LIN {X 0,Y 453.771,Z 399.729,A -85,B 0,C 180,E1 -8336.112,E2 -8336.112} C_VEL
LIN {X 0,Y 453.536,Z 405.266,A -85,B 0,C 180,E1 -8339.245,E2 -8339.245} C_VEL
LIN {X 0,Y 453.322,Z 410.802,A -85,B 0,C 180,E1 -8342.283,E2 -8342.283} C_VEL
LIN {X 0,Y 453.088,Z 416.362,A -85,B 0,C 180,E1 -8345.241,E2 -8345.241} C_VEL
LIN {X 0,Y 452.935,Z 422.796,A -85,B 0,C 180,E1 -8348.59,E2 -8348.59} C_VEL
LIN {X 0,Y 452.827,Z 427.078,A -85,B 0,C 180,E1 -8350.768,E2 -8350.768} C_VEL
LIN {X 0,Y 456.144,Z 441.547,A -85,B 0,C 180,E1 -8351.266,E2 -8351.266} C_VEL
LIN {X 0,Y 458.132,Z 452.718,A -85,B 0,C 180,E1 -8351.752,E2 -8351.752} C_VEL
LIN {X 0,Y 457.605,Z 465.932,A -85,B 0,C 180,E1 -8352.373,E2 -8352.373} C_VEL
LIN {X 0,Y 456.876,Z 478.306,A -85,B 0,C 180,E1 -8353.121,E2 -8353.121} C_VEL
LIN {X 0,Y 456.097,Z 491.399,A -85,B 0,C 180,E1 -8354.127,E2 -8354.127} C_VEL
LIN {X 0,Y 455.413,Z 502.092,A -85,B 0,C 180,E1 -8355.134,E2 -8355.134} C_VEL
LIN {X 0,Y 454.609,Z 512.904,A -85,B 0,C 180,E1 -8356.364,E2 -8356.364} C_VEL
LIN {X 0,Y 454.028,Z 522.647,A -85,B 0,C 180,E1 -8357.711,E2 -8357.711} C_VEL
LIN {X 0,Y 453.518,Z 530.73,A -85,B 0,C 180,E1 -8359.057,E2 -8359.057} C_VEL
LIN {X 0,Y 453.072,Z 538.475,A -85,B 0,C 180,E1 -8360.626,E2 -8360.626} C_VEL
LIN {X 0,Y 452.8,Z 543.883,A -85,B 0,C 180,E1 -8361.97,E2 -8361.97} C_VEL
LIN {X 0,Y 452.604,Z 549.57,A -85,B 0,C 180,E1 -8363.76,E2 -8363.76} C_VEL
LIN {X 0,Y 452.588,Z 551.82,A -85,B 0,C 180,E1 -8364.654,E2 -8364.654} C_VEL
LIN {X 0,Y 452.446,Z 555.217,A -85,B 0,C 180,E1 -8366.438,E2 -8366.438} C_VEL
LIN {X 0,Y 452.43,Z 557.227,A -85,B 0,C 180,E1 -8368.22,E2 -8368.22} C_VEL
LIN {X 0,Y 452.405,Z 557.893,A -85,B 0,C 180,E1 -8370,E2 -8370} C_VEL
LIN {X 0,Y 452.43,Z 557.228,A -85,B 0,C 180,E1 -8371.78,E2 -8371.78} C_VEL
LIN {X 0,Y 452.446,Z 555.22,A -85,B 0,C 180,E1 -8373.562,E2 -8373.562} C_VEL
LIN {X 0,Y 452.588,Z 551.822,A -85,B 0,C 180,E1 -8375.346,E2 -8375.346} C_VEL
LIN {X 0,Y 452.665,Z 546.928,A -85,B 0,C 180,E1 -8377.135,E2 -8377.135} C_VEL
LIN {X 0,Y 452.982,Z 540.398,A -85,B 0,C 180,E1 -8378.925,E2 -8378.925} C_VEL
LIN {X 0,Y 453.348,Z 533.13,A -85,B 0,C 180,E1 -8380.495,E2 -8380.495} C_VEL
LIN {X 0,Y 453.985,Z 524.13,A -85,B 0,C 180,E1 -8382.063,E2 -8382.063} C_VEL
LIN {X 0,Y 454.533,Z 514.682,A -85,B 0,C 180,E1 -8383.411,E2 -8383.411} C_VEL
LIN {X 0,Y 455.236,Z 504.222,A -85,B 0,C 180,E1 -8384.643,E2 -8384.643} C_VEL
LIN {X 0,Y 456.004,Z 492.68,A -85,B 0,C 180,E1 -8385.762,E2 -8385.762} C_VEL
LIN {X 0,Y 456.802,Z 479.875,A -85,B 0,C 180,E1 -8386.766,E2 -8386.766} C_VEL
LIN {X 0,Y 457.502,Z 467.239,A -85,B 0,C 180,E1 -8387.553,E2 -8387.553} C_VEL
LIN {X 0,Y 458.065,Z 453.718,A -85,B 0,C 180,E1 -8388.204,E2 -8388.204} C_VEL
LIN {X 0,Y 457.633,Z 449.129,A -85,B 0,C 180,E1 -8388.406,E2 -8388.406} C_VEL
LIN {X 0,Y 454.892,Z 435.812,A -85,B 0,C 180,E1 -8388.948,E2 -8388.948} C_VEL
LIN {X 0,Y 452.825,Z 427.1,A -85,B 0,C 180,E1 -8389.23,E2 -8389.23} C_VEL
LIN {X 0,Y 452.954,Z 421.91,A -85,B 0,C 180,E1 -8391.863,E2 -8391.863} C_VEL
LIN {X 0,Y 453.088,Z 416.355,A -85,B 0,C 180,E1 -8394.759,E2 -8394.759} C_VEL
LIN {X 0,Y 453.322,Z 410.438,A -85,B 0,C 180,E1 -8397.909,E2 -8397.909} C_VEL
LIN {X 0,Y 453.534,Z 405.256,A -85,B 0,C 180,E1 -8400.755,E2 -8400.755} C_VEL
LIN {X 0,Y 453.77,Z 399.716,A -85,B 0,C 180,E1 -8403.888,E2 -8403.888} C_VEL
LIN {X 0,Y 454.058,Z 394.189,A -85,B 0,C 180,E1 -8407.132,E2 -8407.132} C_VEL
LIN {X 0,Y 454.016,Z 390.49,A -85,B 0,C 180,E1 -8409.395,E2 -8409.395} C_VEL
LIN {X 0,Y 453.497,Z 386.625,A -85,B 0,C 180,E1 -8411.938,E2 -8411.938} C_VEL
LIN {X 0,Y 453.485,Z 386.624,A -85,B 0,C 180,E1 -8415.471,E2 -8415.471} C_VEL
LIN {X 0,Y 453.483,Z 386.625,A -85,B 0,C 180,E1 -8418.21,E2 -8418.21} C_VEL
LIN {X 0,Y 453.534,Z 386.618,A -85,B 0,C 180,E1 -8420.787,E2 -8420.787} C_VEL
LIN {X 0,Y 453.459,Z 386.626,A -85,B 0,C 180,E1 -8423.918,E2 -8423.918} C_VEL
LIN {X 0,Y 453.484,Z 386.623,A -85,B 0,C 180,E1 -8427.151,E2 -8427.151} C_VEL
LIN {X 0,Y 453.476,Z 386.623,A -85,B 0,C 180,E1 -8430.268,E2 -8430.268} C_VEL
LIN {X 0,Y 453.506,Z 386.618,A -85,B 0,C 180,E1 -8433.294,E2 -8433.294} C_VEL
LIN {X 0,Y 453.498,Z 386.62,A -85,B 0,C 180,E1 -8436.239,E2 -8436.239} C_VEL
LIN {X 0,Y 453.485,Z 386.624,A -85,B 0,C 180,E1 -8439.118,E2 -8439.118} C_VEL
LIN {X 0,Y 453.514,Z 386.62,A -85,B 0,C 180,E1 -8441.945,E2 -8441.945} C_VEL
LIN {X 0,Y 453.553,Z 386.612,A -85,B 0,C 180,E1 -8444.727,E2 -8444.727} C_VEL
LIN {X 0,Y 453.562,Z 386.613,A -85,B 0,C 180,E1 -8448.379,E2 -8448.379} C_VEL
LIN {X 0,Y 453.654,Z 386.601,A -85,B 0,C 180,E1 -8451.985,E2 -8451.985} C_VEL
LIN {X 0,Y 453.672,Z 386.598,A -85,B 0,C 180,E1 -8454.667,E2 -8454.667} C_VEL
LIN {X 0,Y 453.767,Z 386.586,A -85,B 0,C 180,E1 -8457.337,E2 -8457.337} C_VEL
LIN {X 0,Y 453.826,Z 386.582,A -85,B 0,C 180,E1 -8460,E2 -8460} C_VEL
LIN {X 0,Y 453.746,Z 386.588,A -85,B 0,C 180,E1 -8462.663,E2 -8462.663} C_VEL
LIN {X 0,Y 453.68,Z 386.599,A -85,B 0,C 180,E1 -8466.225,E2 -8466.225} C_VEL
LIN {X 0,Y 453.594,Z 386.607,A -85,B 0,C 180,E1 -8468.913,E2 -8468.913} C_VEL
LIN {X 0,Y 453.565,Z 386.611,A -85,B 0,C 180,E1 -8472.529,E2 -8472.529} C_VEL
LIN {X 0,Y 453.559,Z 386.615,A -85,B 0,C 180,E1 -8476.196,E2 -8476.196} C_VEL
LIN {X 0,Y 453.523,Z 386.617,A -85,B 0,C 180,E1 -8479.041,E2 -8479.041} C_VEL
LIN {X 0,Y 453.479,Z 386.621,A -85,B 0,C 180,E1 -8481.836,E2 -8481.836} C_VEL
LIN {X 0,Y 453.516,Z 386.618,A -85,B 0,C 180,E1 -8484.734,E2 -8484.734} C_VEL
LIN {X 0,Y 453.539,Z 386.615,A -85,B 0,C 180,E1 -8487.961,E2 -8487.961} C_VEL
LIN {X 0,Y 453.467,Z 386.623,A -85,B 0,C 180,E1 -8491.525,E2 -8491.525} C_VEL
LIN {X 0,Y 453.491,Z 386.62,A -85,B 0,C 180,E1 -8494.778,E2 -8494.778} C_VEL
LIN {X 0,Y 453.476,Z 386.621,A -85,B 0,C 180,E1 -8498.311,E2 -8498.311} C_VEL
LIN {X 0,Y 453.495,Z 386.624,A -85,B 0,C 180,E1 -8500.609,E2 -8500.609} C_VEL
LIN {X 0,Y 453.457,Z 386.626,A -85,B 0,C 180,E1 -8503.244,E2 -8503.244} C_VEL
LIN {X 0,Y 453.478,Z 386.625,A -85,B 0,C 180,E1 -8505.78,E2 -8505.78} C_VEL
LIN {X 0,Y 453.483,Z 386.624,A -85,B 0,C 180,E1 -8508.21,E2 -8508.21} C_VEL
LIN {X 0,Y 453.495,Z 386.623,A -85,B 0,C 180,E1 -8509.409,E2 -8509.409} C_VEL
LIN {X 0,Y 453.656,Z 389.524,A -85,B 0,C 180,E1 -8511.707,E2 -8511.707} C_VEL
LIN {X 0,Y 453.659,Z 392.688,A -85,B 0,C 180,E1 -8513.936,E2 -8513.936} C_VEL
LIN {X 0,Y 453.488,Z 397.459,A -85,B 0,C 180,E1 -8517.152,E2 -8517.152} C_VEL
LIN {X 0,Y 453.293,Z 402.218,A -85,B 0,C 180,E1 -8520.255,E2 -8520.255} C_VEL
LIN {X 0,Y 453.095,Z 406.966,A -85,B 0,C 180,E1 -8523.268,E2 -8523.268} C_VEL
LIN {X 0,Y 452.964,Z 411.797,A -85,B 0,C 180,E1 -8526.266,E2 -8526.266} C_VEL
LIN {X 0,Y 452.871,Z 416.447,A -85,B 0,C 180,E1 -8529.088,E2 -8529.088} C_VEL
LIN {X 0,Y 452.778,Z 419.452,A -85,B 0,C 180,E1 -8530.826,E2 -8530.826} C_VEL
LIN {X 0,Y 456.461,Z 434.331,A -85,B 0,C 180,E1 -8531.364,E2 -8531.364} C_VEL
LIN {X 0,Y 458.247,Z 443.537,A -85,B 0,C 180,E1 -8531.772,E2 -8531.772} C_VEL
LIN {X 0,Y 457.714,Z 456.532,A -85,B 0,C 180,E1 -8532.371,E2 -8532.371} C_VEL
LIN {X 0,Y 457.072,Z 469.188,A -85,B 0,C 180,E1 -8533.129,E2 -8533.129} C_VEL
LIN {X 0,Y 456.337,Z 481.08,A -85,B 0,C 180,E1 -8534.021,E2 -8534.021} C_VEL
LIN {X 0,Y 455.633,Z 492.052,A -85,B 0,C 180,E1 -8535.027,E2 -8535.027} C_VEL
LIN {X 0,Y 454.968,Z 501.163,A -85,B 0,C 180,E1 -8536.025,E2 -8536.025} C_VEL
LIN {X 0,Y 454.028,Z 505.44,A -85,B 0,C 180,E1 -8536.526,E2 -8536.526} C_VEL
LIN {X 0,Y 450.81,Z 512.123,A -85,B 0,C 180,E1 -8537.361,E2 -8537.361} C_VEL
LIN {X 0,Y 447.577,Z 518.308,A -85,B 0,C 180,E1 -8538.262,E2 -8538.262} C_VEL
LIN {X 0,Y 446.623,Z 521.791,A -85,B 0,C 180,E1 -8538.863,E2 -8538.863} C_VEL
LIN {X 0,Y 446.142,Z 529.67,A -85,B 0,C 180,E1 -8540.479,E2 -8540.479} C_VEL
LIN {X 0,Y 445.825,Z 535.089,A -85,B 0,C 180,E1 -8541.844,E2 -8541.844} C_VEL
LIN {X 0,Y 445.598,Z 540.786,A -85,B 0,C 180,E1 -8543.661,E2 -8543.661} C_VEL
LIN {X 0,Y 445.549,Z 543.042,A -85,B 0,C 180,E1 -8544.569,E2 -8544.569} C_VEL
LIN {X 0,Y 445.384,Z 546.456,A -85,B 0,C 180,E1 -8546.381,E2 -8546.381} C_VEL
LIN {X 0,Y 445.432,Z 547.638,A -85,B 0,C 180,E1 -8547.287,E2 -8547.287} C_VEL
LIN {X 0,Y 445.313,Z 548.998,A -85,B 0,C 180,E1 -8549.096,E2 -8549.096} C_VEL
LIN {X 0,Y 445.313,Z 549.036,A -85,B 0,C 180,E1 -8550.904,E2 -8550.904} C_VEL
LIN {X 0,Y 445.431,Z 547.746,A -85,B 0,C 180,E1 -8552.713,E2 -8552.713} C_VEL
LIN {X 0,Y 445.418,Z 545.102,A -85,B 0,C 180,E1 -8554.525,E2 -8554.525} C_VEL
LIN {X 0,Y 445.555,Z 542.191,A -85,B 0,C 180,E1 -8555.885,E2 -8555.885} C_VEL
LIN {X 0,Y 445.728,Z 537.005,A -85,B 0,C 180,E1 -8557.702,E2 -8557.702} C_VEL
LIN {X 0,Y 446.002,Z 531.966,A -85,B 0,C 180,E1 -8559.066,E2 -8559.066} C_VEL
LIN {X 0,Y 446.394,Z 524.772,A -85,B 0,C 180,E1 -8560.661,E2 -8560.661} C_VEL
LIN {X 0,Y 447,Z 517.233,A -85,B 0,C 180,E1 -8562.024,E2 -8562.024} C_VEL
LIN {X 0,Y 447.613,Z 507.838,A -85,B 0,C 180,E1 -8563.44,E2 -8563.44} C_VEL
LIN {X 0,Y 448.382,Z 497.215,A -85,B 0,C 180,E1 -8564.756,E2 -8564.756} C_VEL
LIN {X 0,Y 449.168,Z 486.034,A -85,B 0,C 180,E1 -8565.892,E2 -8565.892} C_VEL
LIN {X 0,Y 450.012,Z 473.662,A -85,B 0,C 180,E1 -8566.91,E2 -8566.91} C_VEL
LIN {X 0,Y 450.769,Z 460.742,A -85,B 0,C 180,E1 -8567.759,E2 -8567.759} C_VEL
LIN {X 0,Y 451.384,Z 446.611,A -85,B 0,C 180,E1 -8568.474,E2 -8568.474} C_VEL
LIN {X 0,Y 451.139,Z 442.421,A -85,B 0,C 180,E1 -8568.665,E2 -8568.665} C_VEL
LIN {X 0,Y 448.115,Z 428.898,A -85,B 0,C 180,E1 -8569.258,E2 -8569.258} C_VEL
LIN {X 0,Y 445.714,Z 419.409,A -85,B 0,C 180,E1 -8569.588,E2 -8569.588} C_VEL
LIN {X 0,Y 445.796,Z 415.08,A -85,B 0,C 180,E1 -8572.232,E2 -8572.232} C_VEL
LIN {X 0,Y 445.949,Z 410.338,A -85,B 0,C 180,E1 -8575.183,E2 -8575.183} C_VEL
LIN {X 0,Y 446.12,Z 405.586,A -85,B 0,C 180,E1 -8578.204,E2 -8578.204} C_VEL
LIN {X 0,Y 446.334,Z 400.828,A -85,B 0,C 180,E1 -8581.307,E2 -8581.307} C_VEL
LIN {X 0,Y 446.54,Z 396.061,A -85,B 0,C 180,E1 -8584.513,E2 -8584.513} C_VEL
LIN {X 0,Y 446.672,Z 392.869,A -85,B 0,C 180,E1 -8586.72,E2 -8586.72} C_VEL
LIN {X 0,Y 446.591,Z 388.971,A -85,B 0,C 180,E1 -8589.546,E2 -8589.546} C_VEL
LIN {X 0,Y 446.446,Z 387.504,A -85,B 0,C 180,E1 -8590.92,E2 -8590.92} C_VEL
LIN {X 0,Y 446.426,Z 387.503,A -85,B 0,C 180,E1 -8593.843,E2 -8593.843} C_VEL
LIN {X 0,Y 446.402,Z 387.51,A -85,B 0,C 180,E1 -8596.403,E2 -8596.403} C_VEL
LIN {X 0,Y 446.429,Z 387.503,A -85,B 0,C 180,E1 -8599.082,E2 -8599.082} C_VEL
LIN {X 0,Y 446.43,Z 387.5,A -85,B 0,C 180,E1 -8602.123,E2 -8602.123} C_VEL
LIN {X 0,Y 446.434,Z 387.5,A -85,B 0,C 180,E1 -8605.477,E2 -8605.477} C_VEL
LIN {X 0,Y 446.419,Z 387.501,A -85,B 0,C 180,E1 -8608.7,E2 -8608.7} C_VEL
LIN {X 0,Y 446.487,Z 387.493,A -85,B 0,C 180,E1 -8611.821,E2 -8611.821} C_VEL
LIN {X 0,Y 446.46,Z 387.496,A -85,B 0,C 180,E1 -8614.848,E2 -8614.848} C_VEL
LIN {X 0,Y 446.451,Z 387.497,A -85,B 0,C 180,E1 -8618.245,E2 -8618.245} C_VEL
LIN {X 0,Y 446.46,Z 387.496,A -85,B 0,C 180,E1 -8621.649,E2 -8621.649} C_VEL
LIN {X 0,Y 446.512,Z 387.489,A -85,B 0,C 180,E1 -8624.48,E2 -8624.48} C_VEL
LIN {X 0,Y 446.521,Z 387.489,A -85,B 0,C 180,E1 -8628.193,E2 -8628.193} C_VEL
LIN {X 0,Y 446.604,Z 387.481,A -85,B 0,C 180,E1 -8631.858,E2 -8631.858} C_VEL
LIN {X 0,Y 446.648,Z 387.473,A -85,B 0,C 180,E1 -8634.583,E2 -8634.583} C_VEL
LIN {X 0,Y 446.667,Z 387.473,A -85,B 0,C 180,E1 -8638.197,E2 -8638.197} C_VEL
LIN {X 0,Y 446.796,Z 387.459,A -85,B 0,C 180,E1 -8640,E2 -8640} C_VEL
LIN {X 0,Y 446.712,Z 387.465,A -85,B 0,C 180,E1 -8642.705,E2 -8642.705} C_VEL
LIN {X 0,Y 446.65,Z 387.474,A -85,B 0,C 180,E1 -8646.324,E2 -8646.324} C_VEL
LIN {X 0,Y 446.541,Z 387.486,A -85,B 0,C 180,E1 -8649.055,E2 -8649.055} C_VEL
LIN {X 0,Y 446.524,Z 387.49,A -85,B 0,C 180,E1 -8652.73,E2 -8652.73} C_VEL
LIN {X 0,Y 446.499,Z 387.496,A -85,B 0,C 180,E1 -8656.228,E2 -8656.228} C_VEL
LIN {X 0,Y 446.472,Z 387.497,A -85,B 0,C 180,E1 -8659.303,E2 -8659.303} C_VEL
LIN {X 0,Y 446.421,Z 387.501,A -85,B 0,C 180,E1 -8662.199,E2 -8662.199} C_VEL
LIN {X 0,Y 446.46,Z 387.495,A -85,B 0,C 180,E1 -8665.152,E2 -8665.152} C_VEL
LIN {X 0,Y 446.487,Z 387.493,A -85,B 0,C 180,E1 -8668.178,E2 -8668.178} C_VEL
LIN {X 0,Y 446.421,Z 387.501,A -85,B 0,C 180,E1 -8671.775,E2 -8671.775} C_VEL
LIN {X 0,Y 446.433,Z 387.501,A -85,B 0,C 180,E1 -8674.523,E2 -8674.523} C_VEL
LIN {X 0,Y 446.441,Z 387.501,A -85,B 0,C 180,E1 -8678.083,E2 -8678.083} C_VEL
LIN {X 0,Y 446.445,Z 387.502,A -85,B 0,C 180,E1 -8680.92,E2 -8680.92} C_VEL
LIN {X 0,Y 446.402,Z 387.508,A -85,B 0,C 180,E1 -8683.846,E2 -8683.846} C_VEL
LIN {X 0,Y 446.4,Z 387.507,A -85,B 0,C 180,E1 -8686.403,E2 -8686.403} C_VEL
LIN {X 0,Y 446.478,Z 387.622,A -85,B 0,C 180,E1 -8687.948,E2 -8687.948} C_VEL
LIN {X 0,Y 446.962,Z 391.326,A -85,B 0,C 180,E1 -8690.396,E2 -8690.396} C_VEL
LIN {X 0,Y 447.066,Z 394.165,A -85,B 0,C 180,E1 -8692.187,E2 -8692.187} C_VEL
LIN {X 0,Y 446.887,Z 398.592,A -85,B 0,C 180,E1 -8694.863,E2 -8694.863} C_VEL
LIN {X 0,Y 446.592,Z 404.304,A -85,B 0,C 180,E1 -8698.19,E2 -8698.19} C_VEL
LIN {X 0,Y 446.341,Z 408.912,A -85,B 0,C 180,E1 -8700.783,E2 -8700.783} C_VEL
LIN {X 0,Y 446.143,Z 414.552,A -85,B 0,C 180,E1 -8703.885,E2 -8703.885} C_VEL
LIN {X 0,Y 445.927,Z 420.003,A -85,B 0,C 180,E1 -8706.796,E2 -8706.796} C_VEL
LIN {X 0,Y 445.775,Z 425.561,A -85,B 0,C 180,E1 -8709.705,E2 -8709.705} C_VEL
LIN {X 0,Y 445.74,Z 426.994,A -85,B 0,C 180,E1 -8710.448,E2 -8710.448} C_VEL
LIN {X 0,Y 449.191,Z 441.706,A -85,B 0,C 180,E1 -8710.972,E2 -8710.972} C_VEL
LIN {X 0,Y 451.23,Z 452.133,A -85,B 0,C 180,E1 -8711.44,E2 -8711.44} C_VEL
LIN {X 0,Y 450.866,Z 464.885,A -85,B 0,C 180,E1 -8712.044,E2 -8712.044} C_VEL
LIN {X 0,Y 450.07,Z 478.24,A -85,B 0,C 180,E1 -8712.858,E2 -8712.858} C_VEL
LIN {X 0,Y 449.224,Z 491.333,A -85,B 0,C 180,E1 -8713.877,E2 -8713.877} C_VEL
LIN {X 0,Y 448.446,Z 503.096,A -85,B 0,C 180,E1 -8715.014,E2 -8715.014} C_VEL
LIN {X 0,Y 447.688,Z 512.837,A -85,B 0,C 180,E1 -8716.149,E2 -8716.149} C_VEL
LIN {X 0,Y 447.022,Z 522.579,A -85,B 0,C 180,E1 -8717.515,E2 -8717.515} C_VEL
LIN {X 0,Y 446.528,Z 530.662,A -85,B 0,C 180,E1 -8718.883,E2 -8718.883} C_VEL
LIN {X 0,Y 446.021,Z 538.407,A -85,B 0,C 180,E1 -8720.477,E2 -8720.477} C_VEL
LIN {X 0,Y 445.741,Z 543.814,A -85,B 0,C 180,E1 -8721.842,E2 -8721.842} C_VEL
LIN {X 0,Y 445.529,Z 549.502,A -85,B 0,C 180,E1 -8723.66,E2 -8723.66} C_VEL
LIN {X 0,Y 445.402,Z 553.628,A -85,B 0,C 180,E1 -8725.475,E2 -8725.475} C_VEL
LIN {X 0,Y 445.394,Z 556.323,A -85,B 0,C 180,E1 -8727.287,E2 -8727.287} C_VEL
LIN {X 0,Y 445.313,Z 557.658,A -85,B 0,C 180,E1 -8729.096,E2 -8729.096} C_VEL
LIN {X 0,Y 445.313,Z 557.658,A -85,B 0,C 180,E1 -8730.904,E2 -8730.904} C_VEL
LIN {X 0,Y 445.394,Z 556.325,A -85,B 0,C 180,E1 -8732.713,E2 -8732.713} C_VEL
LIN {X 0,Y 445.401,Z 553.631,A -85,B 0,C 180,E1 -8734.525,E2 -8734.525} C_VEL
LIN {X 0,Y 445.577,Z 549.5,A -85,B 0,C 180,E1 -8736.339,E2 -8736.339} C_VEL
LIN {X 0,Y 445.74,Z 543.809,A -85,B 0,C 180,E1 -8738.158,E2 -8738.158} C_VEL
LIN {X 0,Y 446.115,Z 537.394,A -85,B 0,C 180,E1 -8739.75,E2 -8739.75} C_VEL
LIN {X 0,Y 446.634,Z 529.422,A -85,B 0,C 180,E1 -8741.344,E2 -8741.344} C_VEL
LIN {X 0,Y 447.171,Z 520.367,A -85,B 0,C 180,E1 -8742.822,E2 -8742.822} C_VEL
LIN {X 0,Y 447.816,Z 511.042,A -85,B 0,C 180,E1 -8744.079,E2 -8744.079} C_VEL
LIN {X 0,Y 448.631,Z 499.842,A -85,B 0,C 180,E1 -8745.329,E2 -8745.329} C_VEL
LIN {X 0,Y 449.542,Z 487.274,A -85,B 0,C 180,E1 -8746.461,E2 -8746.461} C_VEL
LIN {X 0,Y 450.342,Z 474.082,A -85,B 0,C 180,E1 -8747.412,E2 -8747.412} C_VEL
LIN {X 0,Y 451.012,Z 460.834,A -85,B 0,C 180,E1 -8748.159,E2 -8748.159} C_VEL
LIN {X 0,Y 451.187,Z 451.989,A -85,B 0,C 180,E1 -8748.565,E2 -8748.565} C_VEL
LIN {X 0,Y 448.326,Z 437.805,A -85,B 0,C 180,E1 -8749.182,E2 -8749.182} C_VEL
LIN {X 0,Y 445.77,Z 426.99,A -85,B 0,C 180,E1 -8749.55,E2 -8749.55} C_VEL
LIN {X 0,Y 445.901,Z 421.853,A -85,B 0,C 180,E1 -8752.227,E2 -8752.227} C_VEL
LIN {X 0,Y 446.041,Z 416.294,A -85,B 0,C 180,E1 -8755.177,E2 -8755.177} C_VEL
LIN {X 0,Y 446.269,Z 410.743,A -85,B 0,C 180,E1 -8758.193,E2 -8758.193} C_VEL
LIN {X 0,Y 446.534,Z 405.202,A -85,B 0,C 180,E1 -8761.291,E2 -8761.291} C_VEL
LIN {X 0,Y 446.81,Z 399.671,A -85,B 0,C 180,E1 -8764.489,E2 -8764.489} C_VEL
LIN {X 0,Y 447.007,Z 395.986,A -85,B 0,C 180,E1 -8766.694,E2 -8766.694} C_VEL
LIN {X 0,Y 447.022,Z 392.3,A -85,B 0,C 180,E1 -8768.967,E2 -8768.967} C_VEL
LIN {X 0,Y 446.638,Z 388.621,A -85,B 0,C 180,E1 -8771.367,E2 -8771.367} C_VEL
LIN {X 0,Y 446.447,Z 387.503,A -85,B 0,C 180,E1 -8772.279,E2 -8772.279} C_VEL
LIN {X 0,Y 446.452,Z 387.501,A -85,B 0,C 180,E1 -8775.104,E2 -8775.104} C_VEL
LIN {X 0,Y 446.436,Z 387.501,A -85,B 0,C 180,E1 -8778.61,E2 -8778.61} C_VEL
LIN {X 0,Y 446.477,Z 387.498,A -85,B 0,C 180,E1 -8780.976,E2 -8780.976} C_VEL
LIN {X 0,Y 446.423,Z 387.506,A -85,B 0,C 180,E1 -8784.374,E2 -8784.374} C_VEL
LIN {X 0,Y 446.423,Z 387.505,A -85,B 0,C 180,E1 -8787.639,E2 -8787.639} C_VEL
LIN {X 0,Y 446.45,Z 387.502,A -85,B 0,C 180,E1 -8790.791,E2 -8790.791} C_VEL
LIN {X 0,Y 446.479,Z 387.497,A -85,B 0,C 180,E1 -8793.849,E2 -8793.849} C_VEL
LIN {X 0,Y 446.427,Z 387.501,A -85,B 0,C 180,E1 -8796.823,E2 -8796.823} C_VEL
LIN {X 0,Y 446.446,Z 387.497,A -85,B 0,C 180,E1 -8799.737,E2 -8799.737} C_VEL
LIN {X 0,Y 446.467,Z 387.496,A -85,B 0,C 180,E1 -8802.597,E2 -8802.597} C_VEL
LIN {X 0,Y 446.477,Z 387.496,A -85,B 0,C 180,E1 -8805.413,E2 -8805.413} C_VEL
LIN {X 0,Y 446.52,Z 387.489,A -85,B 0,C 180,E1 -8808.193,E2 -8808.193} C_VEL
LIN {X 0,Y 446.602,Z 387.481,A -85,B 0,C 180,E1 -8811.858,E2 -8811.858} C_VEL
LIN {X 0,Y 446.647,Z 387.473,A -85,B 0,C 180,E1 -8814.583,E2 -8814.583} C_VEL
LIN {X 0,Y 446.711,Z 387.465,A -85,B 0,C 180,E1 -8817.295,E2 -8817.295} C_VEL
LIN {X 0,Y 446.796,Z 387.458,A -85,B 0,C 180,E1 -8820,E2 -8820} C_VEL
LIN {X 0,Y 446.693,Z 387.467,A -85,B 0,C 180,E1 -8822.705,E2 -8822.705} C_VEL
LIN {X 0,Y 446.649,Z 387.476,A -85,B 0,C 180,E1 -8826.324,E2 -8826.324} C_VEL
LIN {X 0,Y 446.54,Z 387.486,A -85,B 0,C 180,E1 -8829.055,E2 -8829.055} C_VEL
LIN {X 0,Y 446.523,Z 387.49,A -85,B 0,C 180,E1 -8832.73,E2 -8832.73} C_VEL
LIN {X 0,Y 446.521,Z 387.491,A -85,B 0,C 180,E1 -8836.238,E2 -8836.238} C_VEL
LIN {X 0,Y 446.472,Z 387.498,A -85,B 0,C 180,E1 -8839.303,E2 -8839.303} C_VEL
LIN {X 0,Y 446.42,Z 387.501,A -85,B 0,C 180,E1 -8842.2,E2 -8842.2} C_VEL
LIN {X 0,Y 446.46,Z 387.496,A -85,B 0,C 180,E1 -8845.152,E2 -8845.152} C_VEL
LIN {X 0,Y 446.486,Z 387.493,A -85,B 0,C 180,E1 -8848.179,E2 -8848.179} C_VEL
LIN {X 0,Y 446.421,Z 387.501,A -85,B 0,C 180,E1 -8851.775,E2 -8851.775} C_VEL
LIN {X 0,Y 446.433,Z 387.5,A -85,B 0,C 180,E1 -8854.523,E2 -8854.523} C_VEL
LIN {X 0,Y 446.433,Z 387.498,A -85,B 0,C 180,E1 -8858.082,E2 -8858.082} C_VEL
LIN {X 0,Y 446.428,Z 387.502,A -85,B 0,C 180,E1 -8860.918,E2 -8860.918} C_VEL
LIN {X 0,Y 446.403,Z 387.505,A -85,B 0,C 180,E1 -8863.846,E2 -8863.846} C_VEL
LIN {X 0,Y 446.426,Z 387.502,A -85,B 0,C 180,E1 -8866.4,E2 -8866.4} C_VEL
LIN {X 0,Y 446.429,Z 387.504,A -85,B 0,C 180,E1 -8869.082,E2 -8869.082} C_VEL
LIN {X 0,Y 446.496,Z 387.972,A -85,B 0,C 180,E1 -8869.808,E2 -8869.808} C_VEL
LIN {X 0,Y 446.687,Z 391.143,A -85,B 0,C 180,E1 -8872.149,E2 -8872.149} C_VEL
LIN {X 0,Y 446.568,Z 395.093,A -85,B 0,C 180,E1 -8874.922,E2 -8874.922} C_VEL
LIN {X 0,Y 446.408,Z 399.096,A -85,B 0,C 180,E1 -8877.637,E2 -8877.637} C_VEL
LIN {X 0,Y 446.172,Z 403.851,A -85,B 0,C 180,E1 -8880.771,E2 -8880.771} C_VEL
LIN {X 0,Y 446.035,Z 408.754,A -85,B 0,C 180,E1 -8883.913,E2 -8883.913} C_VEL
LIN {X 0,Y 445.861,Z 413.353,A -85,B 0,C 180,E1 -8886.792,E2 -8886.792} C_VEL
LIN {X 0,Y 445.728,Z 418.09,A -85,B 0,C 180,E1 -8889.703,E2 -8889.703} C_VEL
LIN {X 0,Y 445.725,Z 419.402,A -85,B 0,C 180,E1 -8890.502,E2 -8890.502} C_VEL
LIN {X 0,Y 449.575,Z 434.961,A -85,B 0,C 180,E1 -8891.085,E2 -8891.085} C_VEL
LIN {X 0,Y 451.397,Z 443.728,A -85,B 0,C 180,E1 -8891.49,E2 -8891.49} C_VEL
LIN {X 0,Y 450.902,Z 457.408,A -85,B 0,C 180,E1 -8892.142,E2 -8892.142} C_VEL
LIN {X 0,Y 450.172,Z 470.844,A -85,B 0,C 180,E1 -8892.979,E2 -8892.979} C_VEL
LIN {X 0,Y 449.302,Z 483.733,A -85,B 0,C 180,E1 -8893.997,E2 -8893.997} C_VEL
LIN {X 0,Y 448.488,Z 495.328,A -85,B 0,C 180,E1 -8895.131,E2 -8895.131} C_VEL
LIN {X 0,Y 447.707,Z 505.824,A -85,B 0,C 180,E1 -8896.381,E2 -8896.381} C_VEL
LIN {X 0,Y 447.144,Z 515.293,A -85,B 0,C 180,E1 -8897.75,E2 -8897.75} C_VEL
LIN {X 0,Y 446.623,Z 521.791,A -85,B 0,C 180,E1 -8898.863,E2 -8898.863} C_VEL
LIN {X 0,Y 445.682,Z 525.125,A -85,B 0,C 180,E1 -8899.481,E2 -8899.481} C_VEL
LIN {X 0,Y 442.519,Z 530.199,A -85,B 0,C 180,E1 -8900.502,E2 -8900.502} C_VEL
LIN {X 0,Y 439.45,Z 534.703,A -85,B 0,C 180,E1 -8901.579,E2 -8901.579} C_VEL
LIN {X 0,Y 438.667,Z 537.093,A -85,B 0,C 180,E1 -8902.278,E2 -8902.278} C_VEL
LIN {X 0,Y 438.5,Z 541.624,A -85,B 0,C 180,E1 -8903.845,E2 -8903.845} C_VEL
LIN {X 0,Y 438.347,Z 544.997,A -85,B 0,C 180,E1 -8905.402,E2 -8905.402} C_VEL
LIN {X 0,Y 438.34,Z 547.707,A -85,B 0,C 180,E1 -8907.243,E2 -8907.243} C_VEL
LIN {X 0,Y 438.229,Z 549.067,A -85,B 0,C 180,E1 -8909.081,E2 -8909.081} C_VEL
LIN {X 0,Y 438.229,Z 549.104,A -85,B 0,C 180,E1 -8910.919,E2 -8910.919} C_VEL
LIN {X 0,Y 438.34,Z 547.815,A -85,B 0,C 180,E1 -8912.757,E2 -8912.757} C_VEL
LIN {X 0,Y 438.345,Z 545.17,A -85,B 0,C 180,E1 -8914.598,E2 -8914.598} C_VEL
LIN {X 0,Y 438.506,Z 541.101,A -85,B 0,C 180,E1 -8916.442,E2 -8916.442} C_VEL
LIN {X 0,Y 438.759,Z 535.479,A -85,B 0,C 180,E1 -8918.289,E2 -8918.289} C_VEL
LIN {X 0,Y 439.157,Z 529.132,A -85,B 0,C 180,E1 -8919.906,E2 -8919.906} C_VEL
LIN {X 0,Y 439.731,Z 521.239,A -85,B 0,C 180,E1 -8921.524,E2 -8921.524} C_VEL
LIN {X 0,Y 440.32,Z 512.281,A -85,B 0,C 180,E1 -8923.023,E2 -8923.023} C_VEL
LIN {X 0,Y 441.018,Z 503.036,A -85,B 0,C 180,E1 -8924.301,E2 -8924.301} C_VEL
LIN {X 0,Y 441.869,Z 491.963,A -85,B 0,C 180,E1 -8925.569,E2 -8925.569} C_VEL
LIN {X 0,Y 442.698,Z 480.938,A -85,B 0,C 180,E1 -8926.604,E2 -8926.604} C_VEL
LIN {X 0,Y 443.61,Z 467.75,A -85,B 0,C 180,E1 -8927.602,E2 -8927.602} C_VEL
LIN {X 0,Y 444.277,Z 455.236,A -85,B 0,C 180,E1 -8928.352,E2 -8928.352} C_VEL
LIN {X 0,Y 444.534,Z 444.419,A -85,B 0,C 180,E1 -8928.873,E2 -8928.873} C_VEL
LIN {X 0,Y 441.534,Z 430.703,A -85,B 0,C 180,E1 -8929.509,E2 -8929.509} C_VEL
LIN {X 0,Y 438.655,Z 419.445,A -85,B 0,C 180,E1 -8929.936,E2 -8929.936} C_VEL
LIN {X 0,Y 438.812,Z 413.565,A -85,B 0,C 180,E1 -8933.603,E2 -8933.603} C_VEL
LIN {X 0,Y 438.995,Z 408.807,A -85,B 0,C 180,E1 -8936.632,E2 -8936.632} C_VEL
LIN {X 0,Y 439.159,Z 404.052,A -85,B 0,C 180,E1 -8939.743,E2 -8939.743} C_VEL
LIN {X 0,Y 439.385,Z 399.293,A -85,B 0,C 180,E1 -8942.945,E2 -8942.945} C_VEL
LIN {X 0,Y 439.591,Z 394.503,A -85,B 0,C 180,E1 -8946.267,E2 -8946.267} C_VEL
LIN {X 0,Y 439.602,Z 391.321,A -85,B 0,C 180,E1 -8948.572,E2 -8948.572} C_VEL
LIN {X 0,Y 439.399,Z 388.382,A -85,B 0,C 180,E1 -8950.979,E2 -8950.979} C_VEL
LIN {X 0,Y 439.387,Z 388.38,A -85,B 0,C 180,E1 -8953.964,E2 -8953.964} C_VEL
LIN {X 0,Y 439.354,Z 388.387,A -85,B 0,C 180,E1 -8956.541,E2 -8956.541} C_VEL
LIN {X 0,Y 439.383,Z 388.381,A -85,B 0,C 180,E1 -8959.019,E2 -8959.019} C_VEL
LIN {X 0,Y 439.387,Z 388.378,A -85,B 0,C 180,E1 -8961.606,E2 -8961.606} C_VEL
LIN {X 0,Y 439.404,Z 388.376,A -85,B 0,C 180,E1 -8964.844,E2 -8964.844} C_VEL
LIN {X 0,Y 439.376,Z 388.379,A -85,B 0,C 180,E1 -8968.14,E2 -8968.14} C_VEL
LIN {X 0,Y 439.435,Z 388.371,A -85,B 0,C 180,E1 -8971.598,E2 -8971.598} C_VEL
LIN {X 0,Y 439.408,Z 388.376,A -85,B 0,C 180,E1 -8974.415,E2 -8974.415} C_VEL
LIN {X 0,Y 439.368,Z 388.384,A -85,B 0,C 180,E1 -8977.425,E2 -8977.425} C_VEL
LIN {X 0,Y 439.444,Z 388.373,A -85,B 0,C 180,E1 -8980.663,E2 -8980.663} C_VEL
LIN {X 0,Y 439.466,Z 388.368,A -85,B 0,C 180,E1 -8984.225,E2 -8984.225} C_VEL
LIN {X 0,Y 439.487,Z 388.365,A -85,B 0,C 180,E1 -8988.001,E2 -8988.001} C_VEL
LIN {X 0,Y 439.551,Z 388.358,A -85,B 0,C 180,E1 -8991.726,E2 -8991.726} C_VEL
LIN {X 0,Y 439.624,Z 388.347,A -85,B 0,C 180,E1 -8994.496,E2 -8994.496} C_VEL
LIN {X 0,Y 439.637,Z 388.348,A -85,B 0,C 180,E1 -8998.168,E2 -8998.168} C_VEL
LIN {X 0,Y 439.765,Z 388.334,A -85,B 0,C 180,E1 -9000,E2 -9000} C_VEL
LIN {X 0,Y 439.658,Z 388.344,A -85,B 0,C 180,E1 -9002.749,E2 -9002.749} C_VEL
LIN {X 0,Y 439.621,Z 388.351,A -85,B 0,C 180,E1 -9006.425,E2 -9006.425} C_VEL
LIN {X 0,Y 439.502,Z 388.363,A -85,B 0,C 180,E1 -9009.202,E2 -9009.202} C_VEL
LIN {X 0,Y 439.469,Z 388.37,A -85,B 0,C 180,E1 -9012.937,E2 -9012.937} C_VEL
LIN {X 0,Y 439.45,Z 388.372,A -85,B 0,C 180,E1 -9016.349,E2 -9016.349} C_VEL
LIN {X 0,Y 439.406,Z 388.378,A -85,B 0,C 180,E1 -9019.626,E2 -9019.626} C_VEL
LIN {X 0,Y 439.368,Z 388.383,A -85,B 0,C 180,E1 -9022.575,E2 -9022.575} C_VEL
LIN {X 0,Y 439.408,Z 388.375,A -85,B 0,C 180,E1 -9025.585,E2 -9025.585} C_VEL
LIN {X 0,Y 439.42,Z 388.373,A -85,B 0,C 180,E1 -9028.673,E2 -9028.673} C_VEL
LIN {X 0,Y 439.372,Z 388.38,A -85,B 0,C 180,E1 -9032.03,E2 -9032.03} C_VEL
LIN {X 0,Y 439.399,Z 388.378,A -85,B 0,C 180,E1 -9035.341,E2 -9035.341} C_VEL
LIN {X 0,Y 439.402,Z 388.38,A -85,B 0,C 180,E1 -9038.593,E2 -9038.593} C_VEL
LIN {X 0,Y 439.4,Z 388.378,A -85,B 0,C 180,E1 -9041.258,E2 -9041.258} C_VEL
LIN {X 0,Y 439.401,Z 388.377,A -85,B 0,C 180,E1 -9044.729,E2 -9044.729} C_VEL
LIN {X 0,Y 439.411,Z 388.45,A -85,B 0,C 180,E1 -9047.692,E2 -9047.692} C_VEL
LIN {X 0,Y 439.934,Z 392.285,A -85,B 0,C 180,E1 -9050.282,E2 -9050.282} C_VEL
LIN {X 0,Y 440.006,Z 396.563,A -85,B 0,C 180,E1 -9052.999,E2 -9052.999} C_VEL
LIN {X 0,Y 439.716,Z 401.863,A -85,B 0,C 180,E1 -9056.214,E2 -9056.214} C_VEL
LIN {X 0,Y 439.423,Z 407.007,A -85,B 0,C 180,E1 -9059.216,E2 -9059.216} C_VEL
LIN {X 0,Y 439.183,Z 412.553,A -85,B 0,C 180,E1 -9062.35,E2 -9062.35} C_VEL
LIN {X 0,Y 438.934,Z 418.964,A -85,B 0,C 180,E1 -9065.875,E2 -9065.875} C_VEL
LIN {X 0,Y 438.805,Z 423.649,A -85,B 0,C 180,E1 -9068.385,E2 -9068.385} C_VEL
LIN {X 0,Y 438.704,Z 426.93,A -85,B 0,C 180,E1 -9070.122,E2 -9070.122} C_VEL
LIN {X 0,Y 442.08,Z 441.003,A -85,B 0,C 180,E1 -9070.633,E2 -9070.633} C_VEL
LIN {X 0,Y 444.449,Z 453.348,A -85,B 0,C 180,E1 -9071.204,E2 -9071.204} C_VEL
LIN {X 0,Y 444.068,Z 465.694,A -85,B 0,C 180,E1 -9071.81,E2 -9071.81} C_VEL
LIN {X 0,Y 443.284,Z 478.175,A -85,B 0,C 180,E1 -9072.587,E2 -9072.587} C_VEL
LIN {X 0,Y 442.387,Z 491.267,A -85,B 0,C 180,E1 -9073.621,E2 -9073.621} C_VEL
LIN {X 0,Y 441.536,Z 503.029,A -85,B 0,C 180,E1 -9074.774,E2 -9074.774} C_VEL
LIN {X 0,Y 440.761,Z 512.77,A -85,B 0,C 180,E1 -9075.927,E2 -9075.927} C_VEL
LIN {X 0,Y 440.044,Z 522.511,A -85,B 0,C 180,E1 -9077.314,E2 -9077.314} C_VEL
LIN {X 0,Y 439.542,Z 530.594,A -85,B 0,C 180,E1 -9078.704,E2 -9078.704} C_VEL
LIN {X 0,Y 438.994,Z 538.339,A -85,B 0,C 180,E1 -9080.323,E2 -9080.323} C_VEL
LIN {X 0,Y 438.671,Z 543.746,A -85,B 0,C 180,E1 -9081.71,E2 -9081.71} C_VEL
LIN {X 0,Y 438.447,Z 549.433,A -85,B 0,C 180,E1 -9083.557,E2 -9083.557} C_VEL
LIN {X 0,Y 438.328,Z 553.56,A -85,B 0,C 180,E1 -9085.402,E2 -9085.402} C_VEL
LIN {X 0,Y 438.29,Z 556.254,A -85,B 0,C 180,E1 -9087.243,E2 -9087.243} C_VEL
LIN {X 0,Y 438.228,Z 557.589,A -85,B 0,C 180,E1 -9089.081,E2 -9089.081} C_VEL
LIN {X 0,Y 438.228,Z 557.589,A -85,B 0,C 180,E1 -9090.919,E2 -9090.919} C_VEL
LIN {X 0,Y 438.289,Z 556.256,A -85,B 0,C 180,E1 -9092.757,E2 -9092.757} C_VEL
LIN {X 0,Y 438.327,Z 553.561,A -85,B 0,C 180,E1 -9094.598,E2 -9094.598} C_VEL
LIN {X 0,Y 438.505,Z 549.431,A -85,B 0,C 180,E1 -9096.442,E2 -9096.442} C_VEL
LIN {X 0,Y 438.671,Z 543.739,A -85,B 0,C 180,E1 -9098.29,E2 -9098.29} C_VEL
LIN {X 0,Y 439.093,Z 537.323,A -85,B 0,C 180,E1 -9099.908,E2 -9099.908} C_VEL
LIN {X 0,Y 439.625,Z 529.352,A -85,B 0,C 180,E1 -9101.527,E2 -9101.527} C_VEL
LIN {X 0,Y 440.159,Z 521.012,A -85,B 0,C 180,E1 -9102.917,E2 -9102.917} C_VEL
LIN {X 0,Y 440.882,Z 510.97,A -85,B 0,C 180,E1 -9104.305,E2 -9104.305} C_VEL
LIN {X 0,Y 441.766,Z 499.77,A -85,B 0,C 180,E1 -9105.573,E2 -9105.573} C_VEL
LIN {X 0,Y 442.721,Z 487.202,A -85,B 0,C 180,E1 -9106.722,E2 -9106.722} C_VEL
LIN {X 0,Y 443.549,Z 474.235,A -85,B 0,C 180,E1 -9107.673,E2 -9107.673} C_VEL
LIN {X 0,Y 444.238,Z 460.759,A -85,B 0,C 180,E1 -9108.446,E2 -9108.446} C_VEL
LIN {X 0,Y 444.442,Z 453.301,A -85,B 0,C 180,E1 -9108.795,E2 -9108.795} C_VEL
LIN {X 0,Y 441.681,Z 439.409,A -85,B 0,C 180,E1 -9109.434,E2 -9109.434} C_VEL
LIN {X 0,Y 438.699,Z 426.923,A -85,B 0,C 180,E1 -9109.879,E2 -9109.879} C_VEL
LIN {X 0,Y 438.852,Z 421.781,A -85,B 0,C 180,E1 -9112.603,E2 -9112.603} C_VEL
LIN {X 0,Y 439.008,Z 416.236,A -85,B 0,C 180,E1 -9115.61,E2 -9115.61} C_VEL
LIN {X 0,Y 439.258,Z 410.685,A -85,B 0,C 180,E1 -9118.685,E2 -9118.685} C_VEL
LIN {X 0,Y 439.575,Z 405.157,A -85,B 0,C 180,E1 -9121.844,E2 -9121.844} C_VEL
LIN {X 0,Y 439.886,Z 399.11,A -85,B 0,C 180,E1 -9125.43,E2 -9125.43} C_VEL
LIN {X 0,Y 440.021,Z 395.957,A -85,B 0,C 180,E1 -9127.368,E2 -9127.368} C_VEL
LIN {X 0,Y 439.918,Z 391.945,A -85,B 0,C 180,E1 -9129.93,E2 -9129.93} C_VEL
LIN {X 0,Y 439.403,Z 388.38,A -85,B 0,C 180,E1 -9132.414,E2 -9132.414} C_VEL
LIN {X 0,Y 439.4,Z 388.379,A -85,B 0,C 180,E1 -9135.271,E2 -9135.271} C_VEL
LIN {X 0,Y 439.399,Z 388.378,A -85,B 0,C 180,E1 -9138.742,E2 -9138.742} C_VEL
LIN {X 0,Y 439.395,Z 388.377,A -85,B 0,C 180,E1 -9141.604,E2 -9141.604} C_VEL
LIN {X 0,Y 439.402,Z 388.377,A -85,B 0,C 180,E1 -9144.844,E2 -9144.844} C_VEL
LIN {X 0,Y 439.374,Z 388.38,A -85,B 0,C 180,E1 -9148.14,E2 -9148.14} C_VEL
LIN {X 0,Y 439.433,Z 388.371,A -85,B 0,C 180,E1 -9151.598,E2 -9151.598} C_VEL
LIN {X 0,Y 439.398,Z 388.377,A -85,B 0,C 180,E1 -9154.415,E2 -9154.415} C_VEL
LIN {X 0,Y 439.365,Z 388.383,A -85,B 0,C 180,E1 -9157.425,E2 -9157.425} C_VEL
LIN {X 0,Y 439.443,Z 388.373,A -85,B 0,C 180,E1 -9160.663,E2 -9160.663} C_VEL
LIN {X 0,Y 439.478,Z 388.366,A -85,B 0,C 180,E1 -9164.225,E2 -9164.225} C_VEL
LIN {X 0,Y 439.485,Z 388.364,A -85,B 0,C 180,E1 -9168.001,E2 -9168.001} C_VEL
LIN {X 0,Y 439.55,Z 388.36,A -85,B 0,C 180,E1 -9171.726,E2 -9171.726} C_VEL
LIN {X 0,Y 439.623,Z 388.347,A -85,B 0,C 180,E1 -9174.496,E2 -9174.496} C_VEL
LIN {X 0,Y 439.638,Z 388.348,A -85,B 0,C 180,E1 -9178.168,E2 -9178.168} C_VEL
LIN {X 0,Y 439.766,Z 388.333,A -85,B 0,C 180,E1 -9180,E2 -9180} C_VEL
LIN {X 0,Y 439.642,Z 388.345,A -85,B 0,C 180,E1 -9182.749,E2 -9182.749} C_VEL
LIN {X 0,Y 439.62,Z 388.352,A -85,B 0,C 180,E1 -9186.425,E2 -9186.425} C_VEL
LIN {X 0,Y 439.502,Z 388.363,A -85,B 0,C 180,E1 -9189.202,E2 -9189.202} C_VEL
LIN {X 0,Y 439.468,Z 388.369,A -85,B 0,C 180,E1 -9192.938,E2 -9192.938} C_VEL
LIN {X 0,Y 439.462,Z 388.369,A -85,B 0,C 180,E1 -9196.355,E2 -9196.355} C_VEL
LIN {X 0,Y 439.405,Z 388.378,A -85,B 0,C 180,E1 -9199.626,E2 -9199.626} C_VEL
LIN {X 0,Y 439.367,Z 388.383,A -85,B 0,C 180,E1 -9202.575,E2 -9202.575} C_VEL
LIN {X 0,Y 439.407,Z 388.376,A -85,B 0,C 180,E1 -9205.585,E2 -9205.585} C_VEL
LIN {X 0,Y 439.419,Z 388.373,A -85,B 0,C 180,E1 -9208.673,E2 -9208.673} C_VEL
LIN {X 0,Y 439.372,Z 388.38,A -85,B 0,C 180,E1 -9212.031,E2 -9212.031} C_VEL
LIN {X 0,Y 439.398,Z 388.377,A -85,B 0,C 180,E1 -9215.341,E2 -9215.341} C_VEL
LIN {X 0,Y 439.391,Z 388.377,A -85,B 0,C 180,E1 -9218.594,E2 -9218.594} C_VEL
LIN {X 0,Y 439.39,Z 388.377,A -85,B 0,C 180,E1 -9221.257,E2 -9221.257} C_VEL
LIN {X 0,Y 439.404,Z 388.376,A -85,B 0,C 180,E1 -9224.729,E2 -9224.729} C_VEL
LIN {X 0,Y 439.4,Z 388.377,A -85,B 0,C 180,E1 -9227.796,E2 -9227.796} C_VEL
LIN {X 0,Y 439.383,Z 388.382,A -85,B 0,C 180,E1 -9229.02,E2 -9229.02} C_VEL
LIN {X 0,Y 439.519,Z 389.597,A -85,B 0,C 180,E1 -9230.237,E2 -9230.237} C_VEL
LIN {X 0,Y 439.641,Z 393.419,A -85,B 0,C 180,E1 -9233.062,E2 -9233.062} C_VEL
LIN {X 0,Y 439.454,Z 397.99,A -85,B 0,C 180,E1 -9236.265,E2 -9236.265} C_VEL
LIN {X 0,Y 439.258,Z 402.323,A -85,B 0,C 180,E1 -9239.204,E2 -9239.204} C_VEL
LIN {X 0,Y 439.015,Z 407.078,A -85,B 0,C 180,E1 -9242.338,E2 -9242.338} C_VEL
LIN {X 0,Y 438.916,Z 410.248,A -85,B 0,C 180,E1 -9244.385,E2 -9244.385} C_VEL
LIN {X 0,Y 438.756,Z 414.994,A -85,B 0,C 180,E1 -9247.392,E2 -9247.392} C_VEL
LIN {X 0,Y 438.664,Z 419.471,A -85,B 0,C 180,E1 -9250.175,E2 -9250.175} C_VEL
LIN {X 0,Y 442.609,Z 435.229,A -85,B 0,C 180,E1 -9250.782,E2 -9250.782} C_VEL
LIN {X 0,Y 444.59,Z 444.701,A -85,B 0,C 180,E1 -9251.236,E2 -9251.236} C_VEL
LIN {X 0,Y 444.131,Z 457.896,A -85,B 0,C 180,E1 -9251.885,E2 -9251.885} C_VEL
LIN {X 0,Y 443.389,Z 470.919,A -85,B 0,C 180,E1 -9252.711,E2 -9252.711} C_VEL
LIN {X 0,Y 442.469,Z 483.807,A -85,B 0,C 180,E1 -9253.743,E2 -9253.743} C_VEL
LIN {X 0,Y 441.589,Z 495.402,A -85,B 0,C 180,E1 -9254.894,E2 -9254.894} C_VEL
LIN {X 0,Y 440.796,Z 505.896,A -85,B 0,C 180,E1 -9256.163,E2 -9256.163} C_VEL
LIN {X 0,Y 440.172,Z 515.365,A -85,B 0,C 180,E1 -9257.552,E2 -9257.552} C_VEL
LIN {X 0,Y 439.43,Z 524.402,A -85,B 0,C 180,E1 -9259.168,E2 -9259.168} C_VEL
LIN {X 0,Y 438.977,Z 531.677,A -85,B 0,C 180,E1 -9260.787,E2 -9260.787} C_VEL
LIN {X 0,Y 438.667,Z 537.093,A -85,B 0,C 180,E1 -9262.278,E2 -9262.278} C_VEL
LIN {X 0,Y 437.89,Z 539.341,A -85,B 0,C 180,E1 -9262.989,E2 -9262.989} C_VEL
LIN {X 0,Y 434.878,Z 542.517,A -85,B 0,C 180,E1 -9264.159,E2 -9264.159} C_VEL
LIN {X 0,Y 432.376,Z 544.637,A -85,B 0,C 180,E1 -9265.118,E2 -9265.118} C_VEL
LIN {X 0,Y 431.292,Z 545.988,A -85,B 0,C 180,E1 -9265.87,E2 -9265.87} C_VEL
LIN {X 0,Y 431.198,Z 546.373,A -85,B 0,C 180,E1 -9266.126,E2 -9266.126} C_VEL
LIN {X 0,Y 431.236,Z 547.777,A -85,B 0,C 180,E1 -9267.198,E2 -9267.198} C_VEL
LIN {X 0,Y 431.147,Z 549.136,A -85,B 0,C 180,E1 -9269.066,E2 -9269.066} C_VEL
LIN {X 0,Y 431.147,Z 549.173,A -85,B 0,C 180,E1 -9270.934,E2 -9270.934} C_VEL
LIN {X 0,Y 431.236,Z 547.883,A -85,B 0,C 180,E1 -9272.803,E2 -9272.803} C_VEL
LIN {X 0,Y 431.274,Z 545.238,A -85,B 0,C 180,E1 -9274.674,E2 -9274.674} C_VEL
LIN {X 0,Y 431.44,Z 541.168,A -85,B 0,C 180,E1 -9276.548,E2 -9276.548} C_VEL
LIN {X 0,Y 431.718,Z 535.547,A -85,B 0,C 180,E1 -9278.425,E2 -9278.425} C_VEL
LIN {X 0,Y 432.136,Z 529.199,A -85,B 0,C 180,E1 -9280.069,E2 -9280.069} C_VEL
LIN {X 0,Y 432.747,Z 521.306,A -85,B 0,C 180,E1 -9281.713,E2 -9281.713} C_VEL
LIN {X 0,Y 433.315,Z 513.05,A -85,B 0,C 180,E1 -9283.125,E2 -9283.125} C_VEL
LIN {X 0,Y 434.109,Z 503.101,A -85,B 0,C 180,E1 -9284.533,E2 -9284.533} C_VEL
LIN {X 0,Y 435.033,Z 492.028,A -85,B 0,C 180,E1 -9285.82,E2 -9285.82} C_VEL
LIN {X 0,Y 435.887,Z 481.002,A -85,B 0,C 180,E1 -9286.871,E2 -9286.871} C_VEL
LIN {X 0,Y 436.842,Z 467.902,A -85,B 0,C 180,E1 -9287.878,E2 -9287.878} C_VEL
LIN {X 0,Y 437.554,Z 454.859,A -85,B 0,C 180,E1 -9288.668,E2 -9288.668} C_VEL
LIN {X 0,Y 437.783,Z 445.662,A -85,B 0,C 180,E1 -9289.119,E2 -9289.119} C_VEL
LIN {X 0,Y 434.893,Z 432.349,A -85,B 0,C 180,E1 -9289.767,E2 -9289.767} C_VEL
LIN {X 0,Y 431.59,Z 419.525,A -85,B 0,C 180,E1 -9290.268,E2 -9290.268} C_VEL
LIN {X 0,Y 431.776,Z 413.625,A -85,B 0,C 180,E1 -9294.012,E2 -9294.012} C_VEL
LIN {X 0,Y 431.949,Z 408.875,A -85,B 0,C 180,E1 -9297.102,E2 -9297.102} C_VEL
LIN {X 0,Y 432.19,Z 403.801,A -85,B 0,C 180,E1 -9300.474,E2 -9300.474} C_VEL
LIN {X 0,Y 432.384,Z 399.329,A -85,B 0,C 180,E1 -9303.548,E2 -9303.548} C_VEL
LIN {X 0,Y 432.609,Z 394.545,A -85,B 0,C 180,E1 -9306.948,E2 -9306.948} C_VEL
LIN {X 0,Y 432.518,Z 391.356,A -85,B 0,C 180,E1 -9309.325,E2 -9309.325} C_VEL
LIN {X 0,Y 432.397,Z 389.769,A -85,B 0,C 180,E1 -9310.553,E2 -9310.553} C_VEL
LIN {X 0,Y 432.369,Z 389.255,A -85,B 0,C 180,E1 -9311.793,E2 -9311.793} C_VEL
LIN {X 0,Y 432.343,Z 389.26,A -85,B 0,C 180,E1 -9314.346,E2 -9314.346} C_VEL
LIN {X 0,Y 432.323,Z 389.261,A -85,B 0,C 180,E1 -9317.016,E2 -9317.016} C_VEL
LIN {X 0,Y 432.336,Z 389.258,A -85,B 0,C 180,E1 -9319.821,E2 -9319.821} C_VEL
LIN {X 0,Y 432.318,Z 389.26,A -85,B 0,C 180,E1 -9323.023,E2 -9323.023} C_VEL
LIN {X 0,Y 432.362,Z 389.255,A -85,B 0,C 180,E1 -9325.996,E2 -9325.996} C_VEL
LIN {X 0,Y 432.35,Z 389.255,A -85,B 0,C 180,E1 -9329.49,E2 -9329.49} C_VEL
LIN {X 0,Y 432.395,Z 389.249,A -85,B 0,C 180,E1 -9332.928,E2 -9332.928} C_VEL
LIN {X 0,Y 432.374,Z 389.251,A -85,B 0,C 180,E1 -9336.023,E2 -9336.023} C_VEL
LIN {X 0,Y 432.353,Z 389.254,A -85,B 0,C 180,E1 -9339.046,E2 -9339.046} C_VEL
LIN {X 0,Y 432.381,Z 389.253,A -85,B 0,C 180,E1 -9342.011,E2 -9342.011} C_VEL
LIN {X 0,Y 432.4,Z 389.247,A -85,B 0,C 180,E1 -9344.927,E2 -9344.927} C_VEL
LIN {X 0,Y 432.462,Z 389.24,A -85,B 0,C 180,E1 -9347.803,E2 -9347.803} C_VEL
LIN {X 0,Y 432.495,Z 389.236,A -85,B 0,C 180,E1 -9351.59,E2 -9351.59} C_VEL
LIN {X 0,Y 432.6,Z 389.222,A -85,B 0,C 180,E1 -9354.406,E2 -9354.406} C_VEL
LIN {X 0,Y 432.607,Z 389.224,A -85,B 0,C 180,E1 -9358.138,E2 -9358.138} C_VEL
LIN {X 0,Y 432.735,Z 389.21,A -85,B 0,C 180,E1 -9360,E2 -9360} C_VEL
LIN {X 0,Y 432.608,Z 389.222,A -85,B 0,C 180,E1 -9362.793,E2 -9362.793} C_VEL
LIN {X 0,Y 432.576,Z 389.23,A -85,B 0,C 180,E1 -9366.53,E2 -9366.53} C_VEL
LIN {X 0,Y 432.445,Z 389.243,A -85,B 0,C 180,E1 -9369.353,E2 -9369.353} C_VEL
LIN {X 0,Y 432.434,Z 389.246,A -85,B 0,C 180,E1 -9372.803,E2 -9372.803} C_VEL
LIN {X 0,Y 432.415,Z 389.247,A -85,B 0,C 180,E1 -9376.479,E2 -9376.479} C_VEL
LIN {X 0,Y 432.342,Z 389.255,A -85,B 0,C 180,E1 -9379.96,E2 -9379.96} C_VEL
LIN {X 0,Y 432.322,Z 389.257,A -85,B 0,C 180,E1 -9382.964,E2 -9382.964} C_VEL
LIN {X 0,Y 432.367,Z 389.254,A -85,B 0,C 180,E1 -9386.032,E2 -9386.032} C_VEL
LIN {X 0,Y 432.345,Z 389.258,A -85,B 0,C 180,E1 -9389.187,E2 -9389.187} C_VEL
LIN {X 0,Y 432.325,Z 389.261,A -85,B 0,C 180,E1 -9392.443,E2 -9392.443} C_VEL
LIN {X 0,Y 432.348,Z 389.259,A -85,B 0,C 180,E1 -9395.632,E2 -9395.632} C_VEL
LIN {X 0,Y 432.363,Z 389.258,A -85,B 0,C 180,E1 -9398.718,E2 -9398.718} C_VEL
LIN {X 0,Y 432.368,Z 389.256,A -85,B 0,C 180,E1 -9401.793,E2 -9401.793} C_VEL
LIN {X 0,Y 432.335,Z 389.258,A -85,B 0,C 180,E1 -9404.347,E2 -9404.347} C_VEL
LIN {X 0,Y 432.377,Z 389.332,A -85,B 0,C 180,E1 -9407.469,E2 -9407.469} C_VEL
LIN {X 0,Y 432.866,Z 392.61,A -85,B 0,C 180,E1 -9409.737,E2 -9409.737} C_VEL
LIN {X 0,Y 433.003,Z 395.936,A -85,B 0,C 180,E1 -9411.919,E2 -9411.919} C_VEL
LIN {X 0,Y 432.873,Z 399.663,A -85,B 0,C 180,E1 -9414.271,E2 -9414.271} C_VEL
LIN {X 0,Y 432.544,Z 405.258,A -85,B 0,C 180,E1 -9417.661,E2 -9417.661} C_VEL
LIN {X 0,Y 432.231,Z 410.644,A -85,B 0,C 180,E1 -9420.804,E2 -9420.804} C_VEL
LIN {X 0,Y 431.999,Z 416.188,A -85,B 0,C 180,E1 -9423.944,E2 -9423.944} C_VEL
LIN {X 0,Y 431.78,Z 421.733,A -85,B 0,C 180,E1 -9427.005,E2 -9427.005} C_VEL
LIN {X 0,Y 431.648,Z 426.959,A -85,B 0,C 180,E1 -9429.785,E2 -9429.785} C_VEL
LIN {X 0,Y 435.201,Z 441.536,A -85,B 0,C 180,E1 -9430.334,E2 -9430.334} C_VEL
LIN {X 0,Y 437.648,Z 454.362,A -85,B 0,C 180,E1 -9430.951,E2 -9430.951} C_VEL
LIN {X 0,Y 437.278,Z 466.478,A -85,B 0,C 180,E1 -9431.57,E2 -9431.57} C_VEL
LIN {X 0,Y 436.383,Z 479.693,A -85,B 0,C 180,E1 -9432.424,E2 -9432.424} C_VEL
LIN {X 0,Y 435.455,Z 492.494,A -85,B 0,C 180,E1 -9433.473,E2 -9433.473} C_VEL
LIN {X 0,Y 434.578,Z 504.033,A -85,B 0,C 180,E1 -9434.644,E2 -9434.644} C_VEL
LIN {X 0,Y 433.691,Z 514.486,A -85,B 0,C 180,E1 -9435.932,E2 -9435.932} C_VEL
LIN {X 0,Y 432.998,Z 523.932,A -85,B 0,C 180,E1 -9437.343,E2 -9437.343} C_VEL
LIN {X 0,Y 432.444,Z 531.759,A -85,B 0,C 180,E1 -9438.754,E2 -9438.754} C_VEL
LIN {X 0,Y 431.978,Z 538.271,A -85,B 0,C 180,E1 -9440.164,E2 -9440.164} C_VEL
LIN {X 0,Y 431.621,Z 543.678,A -85,B 0,C 180,E1 -9441.573,E2 -9441.573} C_VEL
LIN {X 0,Y 431.375,Z 549.365,A -85,B 0,C 180,E1 -9443.451,E2 -9443.451} C_VEL
LIN {X 0,Y 431.254,Z 553.491,A -85,B 0,C 180,E1 -9445.326,E2 -9445.326} C_VEL
LIN {X 0,Y 431.185,Z 556.186,A -85,B 0,C 180,E1 -9447.197,E2 -9447.197} C_VEL
LIN {X 0,Y 431.146,Z 557.521,A -85,B 0,C 180,E1 -9449.066,E2 -9449.066} C_VEL
LIN {X 0,Y 431.146,Z 557.521,A -85,B 0,C 180,E1 -9450.934,E2 -9450.934} C_VEL
LIN {X 0,Y 431.185,Z 556.187,A -85,B 0,C 180,E1 -9452.803,E2 -9452.803} C_VEL
LIN {X 0,Y 431.254,Z 553.492,A -85,B 0,C 180,E1 -9454.674,E2 -9454.674} C_VEL
LIN {X 0,Y 431.412,Z 549.361,A -85,B 0,C 180,E1 -9456.548,E2 -9456.548} C_VEL
LIN {X 0,Y 431.621,Z 543.669,A -85,B 0,C 180,E1 -9458.427,E2 -9458.427} C_VEL
LIN {X 0,Y 432.056,Z 537.253,A -85,B 0,C 180,E1 -9460.071,E2 -9460.071} C_VEL
LIN {X 0,Y 432.619,Z 529.281,A -85,B 0,C 180,E1 -9461.716,E2 -9461.716} C_VEL
LIN {X 0,Y 433.287,Z 519.899,A -85,B 0,C 180,E1 -9463.292,E2 -9463.292} C_VEL
LIN {X 0,Y 434.107,Z 509,A -85,B 0,C 180,E1 -9464.773,E2 -9464.773} C_VEL
LIN {X 0,Y 434.963,Z 498.525,A -85,B 0,C 180,E1 -9465.943,E2 -9465.943} C_VEL
LIN {X 0,Y 435.883,Z 487.129,A -85,B 0,C 180,E1 -9466.992,E2 -9466.992} C_VEL
LIN {X 0,Y 436.761,Z 474.374,A -85,B 0,C 180,E1 -9467.942,E2 -9467.942} C_VEL
LIN {X 0,Y 437.499,Z 460.685,A -85,B 0,C 180,E1 -9468.74,E2 -9468.74} C_VEL
LIN {X 0,Y 437.607,Z 454.214,A -85,B 0,C 180,E1 -9469.054,E2 -9469.054} C_VEL
LIN {X 0,Y 434.96,Z 440.552,A -85,B 0,C 180,E1 -9469.706,E2 -9469.706} C_VEL
LIN {X 0,Y 431.636,Z 426.804,A -85,B 0,C 180,E1 -9470.243,E2 -9470.243} C_VEL
LIN {X 0,Y 431.781,Z 421.724,A -85,B 0,C 180,E1 -9472.994,E2 -9472.994} C_VEL
LIN {X 0,Y 432.032,Z 415.329,A -85,B 0,C 180,E1 -9476.53,E2 -9476.53} C_VEL
LIN {X 0,Y 432.225,Z 410.632,A -85,B 0,C 180,E1 -9479.196,E2 -9479.196} C_VEL
LIN {X 0,Y 432.548,Z 405.101,A -85,B 0,C 180,E1 -9482.424,E2 -9482.424} C_VEL
LIN {X 0,Y 432.874,Z 399.586,A -85,B 0,C 180,E1 -9485.767,E2 -9485.767} C_VEL
LIN {X 0,Y 433.002,Z 395.917,A -85,B 0,C 180,E1 -9488.081,E2 -9488.081} C_VEL
LIN {X 0,Y 432.823,Z 392.234,A -85,B 0,C 180,E1 -9490.504,E2 -9490.504} C_VEL
LIN {X 0,Y 432.363,Z 389.257,A -85,B 0,C 180,E1 -9492.579,E2 -9492.579} C_VEL
LIN {X 0,Y 432.333,Z 389.26,A -85,B 0,C 180,E1 -9495.665,E2 -9495.665} C_VEL
LIN {X 0,Y 432.368,Z 389.255,A -85,B 0,C 180,E1 -9498.393,E2 -9498.393} C_VEL
LIN {X 0,Y 432.355,Z 389.254,A -85,B 0,C 180,E1 -9501.852,E2 -9501.852} C_VEL
LIN {X 0,Y 432.342,Z 389.256,A -85,B 0,C 180,E1 -9505.323,E2 -9505.323} C_VEL
LIN {X 0,Y 432.322,Z 389.259,A -85,B 0,C 180,E1 -9508.654,E2 -9508.654} C_VEL
LIN {X 0,Y 432.383,Z 389.25,A -85,B 0,C 180,E1 -9511.877,E2 -9511.877} C_VEL
LIN {X 0,Y 432.347,Z 389.254,A -85,B 0,C 180,E1 -9514.999,E2 -9514.999} C_VEL
LIN {X 0,Y 432.359,Z 389.252,A -85,B 0,C 180,E1 -9518.046,E2 -9518.046} C_VEL
LIN {X 0,Y 432.388,Z 389.249,A -85,B 0,C 180,E1 -9521.03,E2 -9521.03} C_VEL
LIN {X 0,Y 432.445,Z 389.244,A -85,B 0,C 180,E1 -9523.962,E2 -9523.962} C_VEL
LIN {X 0,Y 432.461,Z 389.239,A -85,B 0,C 180,E1 -9527.804,E2 -9527.804} C_VEL
LIN {X 0,Y 432.494,Z 389.238,A -85,B 0,C 180,E1 -9531.59,E2 -9531.59} C_VEL
LIN {X 0,Y 432.599,Z 389.222,A -85,B 0,C 180,E1 -9534.406,E2 -9534.406} C_VEL
LIN {X 0,Y 432.608,Z 389.223,A -85,B 0,C 180,E1 -9538.138,E2 -9538.138} C_VEL
LIN {X 0,Y 432.736,Z 389.209,A -85,B 0,C 180,E1 -9540,E2 -9540} C_VEL
LIN {X 0,Y 432.594,Z 389.223,A -85,B 0,C 180,E1 -9542.794,E2 -9542.794} C_VEL
LIN {X 0,Y 432.575,Z 389.229,A -85,B 0,C 180,E1 -9546.53,E2 -9546.53} C_VEL
LIN {X 0,Y 432.444,Z 389.243,A -85,B 0,C 180,E1 -9549.353,E2 -9549.353} C_VEL
LIN {X 0,Y 432.433,Z 389.246,A -85,B 0,C 180,E1 -9552.804,E2 -9552.804} C_VEL
LIN {X 0,Y 432.425,Z 389.244,A -85,B 0,C 180,E1 -9556.484,E2 -9556.484} C_VEL
LIN {X 0,Y 432.341,Z 389.255,A -85,B 0,C 180,E1 -9559.96,E2 -9559.96} C_VEL
LIN {X 0,Y 432.321,Z 389.26,A -85,B 0,C 180,E1 -9562.964,E2 -9562.964} C_VEL
LIN {X 0,Y 432.367,Z 389.255,A -85,B 0,C 180,E1 -9566.032,E2 -9566.032} C_VEL
LIN {X 0,Y 432.345,Z 389.258,A -85,B 0,C 180,E1 -9569.187,E2 -9569.187} C_VEL
LIN {X 0,Y 432.324,Z 389.261,A -85,B 0,C 180,E1 -9572.443,E2 -9572.443} C_VEL
LIN {X 0,Y 432.348,Z 389.258,A -85,B 0,C 180,E1 -9575.632,E2 -9575.632} C_VEL
LIN {X 0,Y 432.353,Z 389.255,A -85,B 0,C 180,E1 -9578.716,E2 -9578.716} C_VEL
LIN {X 0,Y 432.335,Z 389.257,A -85,B 0,C 180,E1 -9581.797,E2 -9581.797} C_VEL
LIN {X 0,Y 432.335,Z 389.257,A -85,B 0,C 180,E1 -9584.347,E2 -9584.347} C_VEL
LIN {X 0,Y 432.327,Z 389.26,A -85,B 0,C 180,E1 -9587.015,E2 -9587.015} C_VEL
LIN {X 0,Y 432.336,Z 389.259,A -85,B 0,C 180,E1 -9588.398,E2 -9588.398} C_VEL
LIN {X 0,Y 432.361,Z 389.634,A -85,B 0,C 180,E1 -9589.444,E2 -9589.444} C_VEL
LIN {X 0,Y 432.592,Z 392.81,A -85,B 0,C 180,E1 -9591.877,E2 -9591.877} C_VEL
LIN {X 0,Y 432.513,Z 396.197,A -85,B 0,C 180,E1 -9594.337,E2 -9594.337} C_VEL
LIN {X 0,Y 432.316,Z 400.784,A -85,B 0,C 180,E1 -9597.556,E2 -9597.556} C_VEL
LIN {X 0,Y 432.069,Z 405.551,A -85,B 0,C 180,E1 -9600.792,E2 -9600.792} C_VEL
LIN {X 0,Y 431.899,Z 410.307,A -85,B 0,C 180,E1 -9603.937,E2 -9603.937} C_VEL
LIN {X 0,Y 431.7,Z 415.057,A -85,B 0,C 180,E1 -9607.001,E2 -9607.001} C_VEL
LIN {X 0,Y 431.61,Z 419.547,A -85,B 0,C 180,E1 -9609.841,E2 -9609.841} C_VEL
LIN {X 0,Y 435.273,Z 433.953,A -85,B 0,C 180,E1 -9610.399,E2 -9610.399} C_VEL
LIN {X 0,Y 437.792,Z 445.766,A -85,B 0,C 180,E1 -9610.98,E2 -9610.98} C_VEL
LIN {X 0,Y 437.377,Z 458.189,A -85,B 0,C 180,E1 -9611.608,E2 -9611.608} C_VEL
LIN {X 0,Y 436.61,Z 470.995,A -85,B 0,C 180,E1 -9612.433,E2 -9612.433} C_VEL
LIN {X 0,Y 435.657,Z 483.881,A -85,B 0,C 180,E1 -9613.482,E2 -9613.482} C_VEL
LIN {X 0,Y 434.742,Z 495.475,A -85,B 0,C 180,E1 -9614.65,E2 -9614.65} C_VEL
LIN {X 0,Y 433.874,Z 505.969,A -85,B 0,C 180,E1 -9615.938,E2 -9615.938} C_VEL
LIN {X 0,Y 433.198,Z 515.438,A -85,B 0,C 180,E1 -9617.349,E2 -9617.349} C_VEL
LIN {X 0,Y 432.435,Z 524.473,A -85,B 0,C 180,E1 -9618.991,E2 -9618.991} C_VEL
LIN {X 0,Y 431.953,Z 531.747,A -85,B 0,C 180,E1 -9620.636,E2 -9620.636} C_VEL
LIN {X 0,Y 431.542,Z 538.282,A -85,B 0,C 180,E1 -9622.514,E2 -9622.514} C_VEL
LIN {X 0,Y 431.395,Z 543.182,A -85,B 0,C 180,E1 -9624.391,E2 -9624.391} C_VEL
LIN {X 0,Y 431.198,Z 546.373,A -85,B 0,C 180,E1 -9626.126,E2 -9626.126} C_VEL
LIN {X 0,Y 430.506,Z 547.499,A -85,B 0,C 180,E1 -9626.892,E2 -9626.892} C_VEL
LIN {X 0,Y 427.62,Z 548.783,A -85,B 0,C 180,E1 -9628.147,E2 -9628.147} C_VEL
LIN {X 0,Y 425.188,Z 549.292,A -85,B 0,C 180,E1 -9629.167,E2 -9629.167} C_VEL
LIN {X 0,Y 424.14,Z 549.382,A -85,B 0,C 180,E1 -9629.958,E2 -9629.958} C_VEL
LIN {X 0,Y 424.052,Z 549.354,A -85,B 0,C 180,E1 -9630.226,E2 -9630.226} C_VEL
LIN {X 0,Y 424.127,Z 548.763,A -85,B 0,C 180,E1 -9631.899,E2 -9631.899} C_VEL
LIN {X 0,Y 424.103,Z 546.801,A -85,B 0,C 180,E1 -9633.801,E2 -9633.801} C_VEL
LIN {X 0,Y 424.286,Z 543.455,A -85,B 0,C 180,E1 -9635.704,E2 -9635.704} C_VEL
LIN {X 0,Y 424.494,Z 538.629,A -85,B 0,C 180,E1 -9637.611,E2 -9637.611} C_VEL
LIN {X 0,Y 424.903,Z 532.168,A -85,B 0,C 180,E1 -9639.521,E2 -9639.521} C_VEL
LIN {X 0,Y 425.39,Z 524.973,A -85,B 0,C 180,E1 -9641.194,E2 -9641.194} C_VEL
LIN {X 0,Y 426.121,Z 517.432,A -85,B 0,C 180,E1 -9642.623,E2 -9642.623} C_VEL
LIN {X 0,Y 426.772,Z 508.38,A -85,B 0,C 180,E1 -9644.058,E2 -9644.058} C_VEL
LIN {X 0,Y 427.755,Z 497.41,A -85,B 0,C 180,E1 -9645.485,E2 -9645.485} C_VEL
LIN {X 0,Y 428.684,Z 486.226,A -85,B 0,C 180,E1 -9646.673,E2 -9646.673} C_VEL
LIN {X 0,Y 429.636,Z 473.85,A -85,B 0,C 180,E1 -9647.738,E2 -9647.738} C_VEL
LIN {X 0,Y 430.531,Z 461.078,A -85,B 0,C 180,E1 -9648.615,E2 -9648.615} C_VEL
LIN {X 0,Y 431.16,Z 447.923,A -85,B 0,C 180,E1 -9649.32,E2 -9649.32} C_VEL
LIN {X 0,Y 428.573,Z 435.194,A -85,B 0,C 180,E1 -9649.975,E2 -9649.975} C_VEL
LIN {X 0,Y 424.963,Z 421.713,A -85,B 0,C 180,E1 -9650.539,E2 -9650.539} C_VEL
LIN {X 0,Y 424.508,Z 419.592,A -85,B 0,C 180,E1 -9650.622,E2 -9650.622} C_VEL
LIN {X 0,Y 424.639,Z 415.268,A -85,B 0,C 180,E1 -9653.404,E2 -9653.404} C_VEL
LIN {X 0,Y 424.893,Z 410.217,A -85,B 0,C 180,E1 -9656.722,E2 -9656.722} C_VEL
LIN {X 0,Y 425.049,Z 405.752,A -85,B 0,C 180,E1 -9659.738,E2 -9659.738} C_VEL
LIN {X 0,Y 425.301,Z 400.964,A -85,B 0,C 180,E1 -9663.047,E2 -9663.047} C_VEL
LIN {X 0,Y 425.482,Z 396.893,A -85,B 0,C 180,E1 -9665.965,E2 -9665.965} C_VEL
LIN {X 0,Y 425.585,Z 394.588,A -85,B 0,C 180,E1 -9667.663,E2 -9667.663} C_VEL
LIN {X 0,Y 425.401,Z 390.853,A -85,B 0,C 180,E1 -9670.539,E2 -9670.539} C_VEL
LIN {X 0,Y 425.312,Z 390.136,A -85,B 0,C 180,E1 -9671.374,E2 -9671.374} C_VEL
LIN {X 0,Y 425.292,Z 390.139,A -85,B 0,C 180,E1 -9674.718,E2 -9674.718} C_VEL
LIN {X 0,Y 425.293,Z 390.139,A -85,B 0,C 180,E1 -9678.042,E2 -9678.042} C_VEL
LIN {X 0,Y 425.315,Z 390.134,A -85,B 0,C 180,E1 -9681.103,E2 -9681.103} C_VEL
LIN {X 0,Y 425.303,Z 390.134,A -85,B 0,C 180,E1 -9684.664,E2 -9684.664} C_VEL
LIN {X 0,Y 425.268,Z 390.136,A -85,B 0,C 180,E1 -9688.073,E2 -9688.073} C_VEL
LIN {X 0,Y 425.334,Z 390.128,A -85,B 0,C 180,E1 -9691.368,E2 -9691.368} C_VEL
LIN {X 0,Y 425.299,Z 390.133,A -85,B 0,C 180,E1 -9694.555,E2 -9694.555} C_VEL
LIN {X 0,Y 425.291,Z 390.135,A -85,B 0,C 180,E1 -9697.661,E2 -9697.661} C_VEL
LIN {X 0,Y 425.365,Z 390.127,A -85,B 0,C 180,E1 -9700.704,E2 -9700.704} C_VEL
LIN {X 0,Y 425.392,Z 390.124,A -85,B 0,C 180,E1 -9703.688,E2 -9703.688} C_VEL
LIN {X 0,Y 425.415,Z 390.118,A -85,B 0,C 180,E1 -9707.598,E2 -9707.598} C_VEL
LIN {X 0,Y 425.446,Z 390.113,A -85,B 0,C 180,E1 -9711.45,E2 -9711.45} C_VEL
LIN {X 0,Y 425.557,Z 390.1,A -85,B 0,C 180,E1 -9714.313,E2 -9714.313} C_VEL
LIN {X 0,Y 425.576,Z 390.099,A -85,B 0,C 180,E1 -9718.107,E2 -9718.107} C_VEL
LIN {X 0,Y 425.704,Z 390.086,A -85,B 0,C 180,E1 -9720,E2 -9720} C_VEL
LIN {X 0,Y 425.559,Z 390.1,A -85,B 0,C 180,E1 -9722.84,E2 -9722.84} C_VEL
LIN {X 0,Y 425.534,Z 390.106,A -85,B 0,C 180,E1 -9726.639,E2 -9726.639} C_VEL
LIN {X 0,Y 425.404,Z 390.121,A -85,B 0,C 180,E1 -9729.509,E2 -9729.509} C_VEL
LIN {X 0,Y 425.396,Z 390.123,A -85,B 0,C 180,E1 -9732.904,E2 -9732.904} C_VEL
LIN {X 0,Y 425.364,Z 390.124,A -85,B 0,C 180,E1 -9736.605,E2 -9736.605} C_VEL
LIN {X 0,Y 425.331,Z 390.131,A -85,B 0,C 180,E1 -9739.636,E2 -9739.636} C_VEL
LIN {X 0,Y 425.31,Z 390.128,A -85,B 0,C 180,E1 -9743.365,E2 -9743.365} C_VEL
LIN {X 0,Y 425.351,Z 390.124,A -85,B 0,C 180,E1 -9746.844,E2 -9746.844} C_VEL
LIN {X 0,Y 425.293,Z 390.131,A -85,B 0,C 180,E1 -9749.719,E2 -9749.719} C_VEL
LIN {X 0,Y 425.284,Z 390.135,A -85,B 0,C 180,E1 -9753.048,E2 -9753.048} C_VEL
LIN {X 0,Y 425.287,Z 390.139,A -85,B 0,C 180,E1 -9755.929,E2 -9755.929} C_VEL
LIN {X 0,Y 425.316,Z 390.136,A -85,B 0,C 180,E1 -9759.046,E2 -9759.046} C_VEL
LIN {X 0,Y 425.317,Z 390.135,A -85,B 0,C 180,E1 -9761.962,E2 -9761.962} C_VEL
LIN {X 0,Y 425.286,Z 390.138,A -85,B 0,C 180,E1 -9765.283,E2 -9765.283} C_VEL
LIN {X 0,Y 425.323,Z 390.26,A -85,B 0,C 180,E1 -9767.272,E2 -9767.272} C_VEL
LIN {X 0,Y 425.878,Z 394.058,A -85,B 0,C 180,E1 -9769.94,E2 -9769.94} C_VEL
LIN {X 0,Y 425.989,Z 397.728,A -85,B 0,C 180,E1 -9772.379,E2 -9772.379} C_VEL
LIN {X 0,Y 425.777,Z 401.398,A -85,B 0,C 180,E1 -9774.709,E2 -9774.709} C_VEL
LIN {X 0,Y 425.458,Z 406.913,A -85,B 0,C 180,E1 -9778.089,E2 -9778.089} C_VEL
LIN {X 0,Y 425.18,Z 412.442,A -85,B 0,C 180,E1 -9781.357,E2 -9781.357} C_VEL
LIN {X 0,Y 424.895,Z 417.967,A -85,B 0,C 180,E1 -9784.529,E2 -9784.529} C_VEL
LIN {X 0,Y 424.655,Z 424.079,A -85,B 0,C 180,E1 -9787.941,E2 -9787.941} C_VEL
LIN {X 0,Y 424.563,Z 426.791,A -85,B 0,C 180,E1 -9789.428,E2 -9789.428} C_VEL
LIN {X 0,Y 428.254,Z 441.797,A -85,B 0,C 180,E1 -9790.013,E2 -9790.013} C_VEL
LIN {X 0,Y 430.821,Z 455.12,A -85,B 0,C 180,E1 -9790.676,E2 -9790.676} C_VEL
LIN {X 0,Y 430.764,Z 461.958,A -85,B 0,C 180,E1 -9791.024,E2 -9791.024} C_VEL
LIN {X 0,Y 429.991,Z 474.468,A -85,B 0,C 180,E1 -9791.773,E2 -9791.773} C_VEL
LIN {X 0,Y 429.08,Z 487.095,A -85,B 0,C 180,E1 -9792.73,E2 -9792.73} C_VEL
LIN {X 0,Y 427.994,Z 499.66,A -85,B 0,C 180,E1 -9793.913,E2 -9793.913} C_VEL
LIN {X 0,Y 427.065,Z 510.852,A -85,B 0,C 180,E1 -9795.222,E2 -9795.222} C_VEL
LIN {X 0,Y 426.233,Z 520.889,A -85,B 0,C 180,E1 -9796.653,E2 -9796.653} C_VEL
LIN {X 0,Y 425.63,Z 529.225,A -85,B 0,C 180,E1 -9798.088,E2 -9798.088} C_VEL
LIN {X 0,Y 424.99,Z 537.193,A -85,B 0,C 180,E1 -9799.76,E2 -9799.76} C_VEL
LIN {X 0,Y 424.584,Z 543.609,A -85,B 0,C 180,E1 -9801.432,E2 -9801.432} C_VEL
LIN {X 0,Y 424.298,Z 549.297,A -85,B 0,C 180,E1 -9803.342,E2 -9803.342} C_VEL
LIN {X 0,Y 424.181,Z 553.423,A -85,B 0,C 180,E1 -9805.248,E2 -9805.248} C_VEL
LIN {X 0,Y 424.082,Z 556.117,A -85,B 0,C 180,E1 -9807.15,E2 -9807.15} C_VEL
LIN {X 0,Y 424.067,Z 557.452,A -85,B 0,C 180,E1 -9809.05,E2 -9809.05} C_VEL
LIN {X 0,Y 424.067,Z 557.452,A -85,B 0,C 180,E1 -9810.95,E2 -9810.95} C_VEL
LIN {X 0,Y 424.082,Z 556.117,A -85,B 0,C 180,E1 -9812.85,E2 -9812.85} C_VEL
LIN {X 0,Y 424.182,Z 553.423,A -85,B 0,C 180,E1 -9814.752,E2 -9814.752} C_VEL
LIN {X 0,Y 424.339,Z 549.291,A -85,B 0,C 180,E1 -9816.658,E2 -9816.658} C_VEL
LIN {X 0,Y 424.584,Z 543.599,A -85,B 0,C 180,E1 -9818.567,E2 -9818.567} C_VEL
LIN {X 0,Y 424.989,Z 537.182,A -85,B 0,C 180,E1 -9820.24,E2 -9820.24} C_VEL
LIN {X 0,Y 425.63,Z 529.21,A -85,B 0,C 180,E1 -9821.911,E2 -9821.911} C_VEL
LIN {X 0,Y 426.285,Z 520.433,A -85,B 0,C 180,E1 -9823.416,E2 -9823.416} C_VEL
LIN {X 0,Y 427.065,Z 510.828,A -85,B 0,C 180,E1 -9824.778,E2 -9824.778} C_VEL
LIN {X 0,Y 428.016,Z 499.626,A -85,B 0,C 180,E1 -9826.086,E2 -9826.086} C_VEL
LIN {X 0,Y 429.086,Z 487.056,A -85,B 0,C 180,E1 -9827.27,E2 -9827.27} C_VEL
LIN {X 0,Y 429.98,Z 474.511,A -85,B 0,C 180,E1 -9828.22,E2 -9828.22} C_VEL
LIN {X 0,Y 430.771,Z 460.61,A -85,B 0,C 180,E1 -9829.044,E2 -9829.044} C_VEL
LIN {X 0,Y 430.793,Z 455.028,A -85,B 0,C 180,E1 -9829.325,E2 -9829.325} C_VEL
LIN {X 0,Y 428.208,Z 441.841,A -85,B 0,C 180,E1 -9829.983,E2 -9829.983} C_VEL
LIN {X 0,Y 424.684,Z 427.635,A -85,B 0,C 180,E1 -9830.541,E2 -9830.541} C_VEL
LIN {X 0,Y 424.574,Z 426.739,A -85,B 0,C 180,E1 -9830.595,E2 -9830.595} C_VEL
LIN {X 0,Y 424.728,Z 421.66,A -85,B 0,C 180,E1 -9833.399,E2 -9833.399} C_VEL
LIN {X 0,Y 424.984,Z 415.722,A -85,B 0,C 180,E1 -9836.747,E2 -9836.747} C_VEL
LIN {X 0,Y 425.247,Z 410.58,A -85,B 0,C 180,E1 -9839.723,E2 -9839.723} C_VEL
LIN {X 0,Y 425.556,Z 405.063,A -85,B 0,C 180,E1 -9843.024,E2 -9843.024} C_VEL
LIN {X 0,Y 425.899,Z 399.545,A -85,B 0,C 180,E1 -9846.445,E2 -9846.445} C_VEL
LIN {X 0,Y 425.963,Z 395.382,A -85,B 0,C 180,E1 -9849.154,E2 -9849.154} C_VEL
LIN {X 0,Y 425.621,Z 392.192,A -85,B 0,C 180,E1 -9851.338,E2 -9851.338} C_VEL
LIN {X 0,Y 425.326,Z 390.133,A -85,B 0,C 180,E1 -9852.82,E2 -9852.82} C_VEL
LIN {X 0,Y 425.262,Z 390.143,A -85,B 0,C 180,E1 -9856.044,E2 -9856.044} C_VEL
LIN {X 0,Y 425.305,Z 390.134,A -85,B 0,C 180,E1 -9858.625,E2 -9858.625} C_VEL
LIN {X 0,Y 425.326,Z 390.133,A -85,B 0,C 180,E1 -9861.104,E2 -9861.104} C_VEL
LIN {X 0,Y 425.302,Z 390.134,A -85,B 0,C 180,E1 -9864.664,E2 -9864.664} C_VEL
LIN {X 0,Y 425.266,Z 390.138,A -85,B 0,C 180,E1 -9868.073,E2 -9868.073} C_VEL
LIN {X 0,Y 425.332,Z 390.129,A -85,B 0,C 180,E1 -9871.368,E2 -9871.368} C_VEL
LIN {X 0,Y 425.355,Z 390.126,A -85,B 0,C 180,E1 -9873.506,E2 -9873.506} C_VEL
LIN {X 0,Y 425.285,Z 390.134,A -85,B 0,C 180,E1 -9876.634,E2 -9876.634} C_VEL
LIN {X 0,Y 425.297,Z 390.132,A -85,B 0,C 180,E1 -9879.695,E2 -9879.695} C_VEL
LIN {X 0,Y 425.345,Z 390.126,A -85,B 0,C 180,E1 -9882.698,E2 -9882.698} C_VEL
LIN {X 0,Y 425.354,Z 390.126,A -85,B 0,C 180,E1 -9885.65,E2 -9885.65} C_VEL
LIN {X 0,Y 425.354,Z 390.127,A -85,B 0,C 180,E1 -9888.564,E2 -9888.564} C_VEL
LIN {X 0,Y 425.539,Z 390.099,A -85,B 0,C 180,E1 -9892.408,E2 -9892.408} C_VEL
LIN {X 0,Y 425.556,Z 390.1,A -85,B 0,C 180,E1 -9894.313,E2 -9894.313} C_VEL
LIN {X 0,Y 425.577,Z 390.099,A -85,B 0,C 180,E1 -9898.107,E2 -9898.107} C_VEL
LIN {X 0,Y 425.705,Z 390.085,A -85,B 0,C 180,E1 -9900,E2 -9900} C_VEL
LIN {X 0,Y 425.548,Z 390.101,A -85,B 0,C 180,E1 -9902.84,E2 -9902.84} C_VEL
LIN {X 0,Y 425.533,Z 390.106,A -85,B 0,C 180,E1 -9906.649,E2 -9906.649} C_VEL
LIN {X 0,Y 425.403,Z 390.121,A -85,B 0,C 180,E1 -9909.509,E2 -9909.509} C_VEL
LIN {X 0,Y 425.395,Z 390.122,A -85,B 0,C 180,E1 -9912.904,E2 -9912.904} C_VEL
LIN {X 0,Y 425.372,Z 390.121,A -85,B 0,C 180,E1 -9916.609,E2 -9916.609} C_VEL
LIN {X 0,Y 425.33,Z 390.131,A -85,B 0,C 180,E1 -9919.636,E2 -9919.636} C_VEL
LIN {X 0,Y 425.309,Z 390.131,A -85,B 0,C 180,E1 -9923.365,E2 -9923.365} C_VEL
LIN {X 0,Y 425.35,Z 390.125,A -85,B 0,C 180,E1 -9926.845,E2 -9926.845} C_VEL
LIN {X 0,Y 425.293,Z 390.133,A -85,B 0,C 180,E1 -9929.72,E2 -9929.72} C_VEL
LIN {X 0,Y 425.284,Z 390.134,A -85,B 0,C 180,E1 -9933.048,E2 -9933.048} C_VEL
LIN {X 0,Y 425.287,Z 390.137,A -85,B 0,C 180,E1 -9935.929,E2 -9935.929} C_VEL
LIN {X 0,Y 425.302,Z 390.135,A -85,B 0,C 180,E1 -9939.044,E2 -9939.044} C_VEL
LIN {X 0,Y 425.276,Z 390.137,A -85,B 0,C 180,E1 -9942.653,E2 -9942.653} C_VEL
LIN {X 0,Y 425.271,Z 390.138,A -85,B 0,C 180,E1 -9946.045,E2 -9946.045} C_VEL
LIN {X 0,Y 425.281,Z 390.138,A -85,B 0,C 180,E1 -9948.622,E2 -9948.622} C_VEL
LIN {X 0,Y 425.452,Z 391.26,A -85,B 0,C 180,E1 -9949.892,E2 -9949.892} C_VEL
LIN {X 0,Y 425.587,Z 394.58,A -85,B 0,C 180,E1 -9952.435,E2 -9952.435} C_VEL
LIN {X 0,Y 425.414,Z 399.053,A -85,B 0,C 180,E1 -9955.692,E2 -9955.692} C_VEL
LIN {X 0,Y 425.168,Z 404.152,A -85,B 0,C 180,E1 -9959.267,E2 -9959.267} C_VEL
LIN {X 0,Y 424.912,Z 408.782,A -85,B 0,C 180,E1 -9962.412,E2 -9962.412} C_VEL
LIN {X 0,Y 424.724,Z 413.541,A -85,B 0,C 180,E1 -9965.564,E2 -9965.564} C_VEL
LIN {X 0,Y 424.568,Z 418.293,A -85,B 0,C 180,E1 -9968.643,E2 -9968.643} C_VEL
LIN {X 0,Y 424.544,Z 419.638,A -85,B 0,C 180,E1 -9969.491,E2 -9969.491} C_VEL
LIN {X 0,Y 428.334,Z 434.279,A -85,B 0,C 180,E1 -9970.077,E2 -9970.077} C_VEL
LIN {X 0,Y 431.019,Z 446.913,A -85,B 0,C 180,E1 -9970.72,E2 -9970.72} C_VEL
LIN {X 0,Y 430.625,Z 458.265,A -85,B 0,C 180,E1 -9971.309,E2 -9971.309} C_VEL
LIN {X 0,Y 429.833,Z 471.07,A -85,B 0,C 180,E1 -9972.147,E2 -9972.147} C_VEL
LIN {X 0,Y 428.828,Z 483.955,A -85,B 0,C 180,E1 -9973.211,E2 -9973.211} C_VEL
LIN {X 0,Y 427.885,Z 495.548,A -85,B 0,C 180,E1 -9974.398,E2 -9974.398} C_VEL
LIN {X 0,Y 426.962,Z 506.042,A -85,B 0,C 180,E1 -9975.706,E2 -9975.706} C_VEL
LIN {X 0,Y 426.232,Z 515.51,A -85,B 0,C 180,E1 -9977.138,E2 -9977.138} C_VEL
LIN {X 0,Y 425.555,Z 523.357,A -85,B 0,C 180,E1 -9978.57,E2 -9978.57} C_VEL
LIN {X 0,Y 425.058,Z 529.883,A -85,B 0,C 180,E1 -9980.002,E2 -9980.002} C_VEL
LIN {X 0,Y 424.674,Z 535.301,A -85,B 0,C 180,E1 -9981.434,E2 -9981.434} C_VEL
LIN {X 0,Y 424.399,Z 540.996,A -85,B 0,C 180,E1 -9983.343,E2 -9983.343} C_VEL
LIN {X 0,Y 424.208,Z 545.137,A -85,B 0,C 180,E1 -9985.248,E2 -9985.248} C_VEL
LIN {X 0,Y 424.133,Z 547.846,A -85,B 0,C 180,E1 -9987.151,E2 -9987.151} C_VEL
LIN {X 0,Y 424.068,Z 549.205,A -85,B 0,C 180,E1 -9989.05,E2 -9989.05} C_VEL
LIN {X 0,Y 424.052,Z 549.354,A -85,B 0,C 180,E1 -9990.226,E2 -9990.226} C_VEL
LIN {X 0,Y 423.367,Z 549.223,A -85,B 0,C 180,E1 -9991.019,E2 -9991.019} C_VEL
LIN {X 0,Y 420.484,Z 548.478,A -85,B 0,C 180,E1 -9992.306,E2 -9992.306} C_VEL
LIN {X 0,Y 418.092,Z 547.491,A -85,B 0,C 180,E1 -9993.338,E2 -9993.338} C_VEL
LIN {X 0,Y 417.119,Z 546.471,A -85,B 0,C 180,E1 -9994.131,E2 -9994.131} C_VEL
LIN {X 0,Y 417.069,Z 546.047,A -85,B 0,C 180,E1 -9994.397,E2 -9994.397} C_VEL
LIN {X 0,Y 417.285,Z 542.13,A -85,B 0,C 180,E1 -9996.438,E2 -9996.438} C_VEL
LIN {X 0,Y 417.52,Z 537.276,A -85,B 0,C 180,E1 -9998.226,E2 -9998.226} C_VEL
LIN {X 0,Y 417.858,Z 532.235,A -85,B 0,C 180,E1 -9999.683,E2 -9999.683} C_VEL
LIN {X 0,Y 418.408,Z 525.04,A -85,B 0,C 180,E1 -10001.383,E2 -10001.383} C_VEL
LIN {X 0,Y 419.244,Z 516.313,A -85,B 0,C 180,E1 -10003.049,E2 -10003.049} C_VEL
LIN {X 0,Y 420.016,Z 506.789,A -85,B 0,C 180,E1 -10004.536,E2 -10004.536} C_VEL
LIN {X 0,Y 420.966,Z 496.432,A -85,B 0,C 180,E1 -10005.866,E2 -10005.866} C_VEL
LIN {X 0,Y 421.986,Z 485.003,A -85,B 0,C 180,E1 -10007.07,E2 -10007.07} C_VEL
LIN {X 0,Y 422.977,Z 472.334,A -85,B 0,C 180,E1 -10008.152,E2 -10008.152} C_VEL
LIN {X 0,Y 423.857,Z 460.049,A -85,B 0,C 180,E1 -10008.988,E2 -10008.988} C_VEL
LIN {X 0,Y 424.385,Z 448.751,A -85,B 0,C 180,E1 -10009.604,E2 -10009.604} C_VEL
LIN {X 0,Y 421.601,Z 435.362,A -85,B 0,C 180,E1 -10010.316,E2 -10010.316} C_VEL
LIN {X 0,Y 417.864,Z 421.593,A -85,B 0,C 180,E1 -10010.908,E2 -10010.908} C_VEL
LIN {X 0,Y 417.462,Z 419.647,A -85,B 0,C 180,E1 -10010.994,E2 -10010.994} C_VEL
LIN {X 0,Y 417.705,Z 413.747,A -85,B 0,C 180,E1 -10014.875,E2 -10014.875} C_VEL
LIN {X 0,Y 417.878,Z 408.987,A -85,B 0,C 180,E1 -10018.094,E2 -10018.094} C_VEL
LIN {X 0,Y 418.142,Z 404.197,A -85,B 0,C 180,E1 -10021.402,E2 -10021.402} C_VEL
LIN {X 0,Y 418.377,Z 399.732,A -85,B 0,C 180,E1 -10024.602,E2 -10024.602} C_VEL
LIN {X 0,Y 418.535,Z 396.229,A -85,B 0,C 180,E1 -10027.194,E2 -10027.194} C_VEL
LIN {X 0,Y 418.476,Z 393.028,A -85,B 0,C 180,E1 -10029.657,E2 -10029.657} C_VEL
LIN {X 0,Y 418.318,Z 391.438,A -85,B 0,C 180,E1 -10030.937,E2 -10030.937} C_VEL
LIN {X 0,Y 418.25,Z 391.013,A -85,B 0,C 180,E1 -10032.324,E2 -10032.324} C_VEL
LIN {X 0,Y 418.241,Z 391.014,A -85,B 0,C 180,E1 -10035.109,E2 -10035.109} C_VEL
LIN {X 0,Y 418.243,Z 391.017,A -85,B 0,C 180,E1 -10037.767,E2 -10037.767} C_VEL
LIN {X 0,Y 418.261,Z 391.01,A -85,B 0,C 180,E1 -10041.559,E2 -10041.559} C_VEL
LIN {X 0,Y 418.263,Z 391.009,A -85,B 0,C 180,E1 -10045.159,E2 -10045.159} C_VEL
LIN {X 0,Y 418.248,Z 391.014,A -85,B 0,C 180,E1 -10047.472,E2 -10047.472} C_VEL
LIN {X 0,Y 418.271,Z 391.01,A -85,B 0,C 180,E1 -10050.895,E2 -10050.895} C_VEL
LIN {X 0,Y 418.274,Z 391.011,A -85,B 0,C 180,E1 -10054.096,E2 -10054.096} C_VEL
LIN {X 0,Y 418.241,Z 391.013,A -85,B 0,C 180,E1 -10057.264,E2 -10057.264} C_VEL
LIN {X 0,Y 418.286,Z 391.005,A -85,B 0,C 180,E1 -10060.364,E2 -10060.364} C_VEL
LIN {X 0,Y 418.32,Z 391.002,A -85,B 0,C 180,E1 -10063.405,E2 -10063.405} C_VEL
LIN {X 0,Y 418.349,Z 391.001,A -85,B 0,C 180,E1 -10066.999,E2 -10066.999} C_VEL
LIN {X 0,Y 418.344,Z 391.002,A -85,B 0,C 180,E1 -10070.329,E2 -10070.329} C_VEL
LIN {X 0,Y 418.516,Z 390.978,A -85,B 0,C 180,E1 -10072.279,E2 -10072.279} C_VEL
LIN {X 0,Y 418.516,Z 390.977,A -85,B 0,C 180,E1 -10074.217,E2 -10074.217} C_VEL
LIN {X 0,Y 418.545,Z 390.975,A -85,B 0,C 180,E1 -10078.075,E2 -10078.075} C_VEL
LIN {X 0,Y 418.674,Z 390.961,A -85,B 0,C 180,E1 -10080,E2 -10080} C_VEL
LIN {X 0,Y 418.513,Z 390.978,A -85,B 0,C 180,E1 -10082.888,E2 -10082.888} C_VEL
LIN {X 0,Y 418.497,Z 390.982,A -85,B 0,C 180,E1 -10086.751,E2 -10086.751} C_VEL
LIN {X 0,Y 418.36,Z 391,A -85,B 0,C 180,E1 -10089.671,E2 -10089.671} C_VEL
LIN {X 0,Y 418.349,Z 391.001,A -85,B 0,C 180,E1 -10093.001,E2 -10093.001} C_VEL
LIN {X 0,Y 418.316,Z 391.002,A -85,B 0,C 180,E1 -10096.736,E2 -10096.736} C_VEL
LIN {X 0,Y 418.274,Z 391.009,A -85,B 0,C 180,E1 -10099.79,E2 -10099.79} C_VEL
LIN {X 0,Y 418.241,Z 391.013,A -85,B 0,C 180,E1 -10102.736,E2 -10102.736} C_VEL
LIN {X 0,Y 418.274,Z 391.011,A -85,B 0,C 180,E1 -10105.904,E2 -10105.904} C_VEL
LIN {X 0,Y 418.267,Z 391.011,A -85,B 0,C 180,E1 -10109.162,E2 -10109.162} C_VEL
LIN {X 0,Y 418.259,Z 391.011,A -85,B 0,C 180,E1 -10112.844,E2 -10112.844} C_VEL
LIN {X 0,Y 418.251,Z 391.013,A -85,B 0,C 180,E1 -10116.239,E2 -10116.239} C_VEL
LIN {X 0,Y 418.268,Z 391.011,A -85,B 0,C 180,E1 -10119.68,E2 -10119.68} C_VEL
LIN {X 0,Y 418.247,Z 391.015,A -85,B 0,C 180,E1 -10122.323,E2 -10122.323} C_VEL
LIN {X 0,Y 418.237,Z 391.016,A -85,B 0,C 180,E1 -10125.109,E2 -10125.109} C_VEL
LIN {X 0,Y 418.292,Z 391.224,A -85,B 0,C 180,E1 -10127.094,E2 -10127.094} C_VEL
LIN {X 0,Y 418.737,Z 394.017,A -85,B 0,C 180,E1 -10129.113,E2 -10129.113} C_VEL
LIN {X 0,Y 418.951,Z 397.689,A -85,B 0,C 180,E1 -10131.634,E2 -10131.634} C_VEL
LIN {X 0,Y 418.826,Z 401.349,A -85,B 0,C 180,E1 -10134.034,E2 -10134.034} C_VEL
LIN {X 0,Y 418.472,Z 406.866,A -85,B 0,C 180,E1 -10137.491,E2 -10137.491} C_VEL
LIN {X 0,Y 418.157,Z 412.375,A -85,B 0,C 180,E1 -10140.83,E2 -10140.83} C_VEL
LIN {X 0,Y 417.874,Z 417.909,A -85,B 0,C 180,E1 -10144.069,E2 -10144.069} C_VEL
LIN {X 0,Y 417.599,Z 424.396,A -85,B 0,C 180,E1 -10147.763,E2 -10147.763} C_VEL
LIN {X 0,Y 417.537,Z 426.835,A -85,B 0,C 180,E1 -10149.07,E2 -10149.07} C_VEL
LIN {X 0,Y 421.145,Z 441.312,A -85,B 0,C 180,E1 -10149.646,E2 -10149.646} C_VEL
LIN {X 0,Y 423.641,Z 453.82,A -85,B 0,C 180,E1 -10150.276,E2 -10150.276} C_VEL
LIN {X 0,Y 424.192,Z 458.839,A -85,B 0,C 180,E1 -10150.549,E2 -10150.549} C_VEL
LIN {X 0,Y 423.454,Z 471.536,A -85,B 0,C 180,E1 -10151.278,E2 -10151.278} C_VEL
LIN {X 0,Y 422.507,Z 484.176,A -85,B 0,C 180,E1 -10152.203,E2 -10152.203} C_VEL
LIN {X 0,Y 421.479,Z 496.071,A -85,B 0,C 180,E1 -10153.283,E2 -10153.283} C_VEL
LIN {X 0,Y 420.554,Z 506.936,A -85,B 0,C 180,E1 -10154.491,E2 -10154.491} C_VEL
LIN {X 0,Y 419.552,Z 517.671,A -85,B 0,C 180,E1 -10155.943,E2 -10155.943} C_VEL
LIN {X 0,Y 418.84,Z 526.535,A -85,B 0,C 180,E1 -10157.4,E2 -10157.4} C_VEL
LIN {X 0,Y 418.12,Z 535.028,A -85,B 0,C 180,E1 -10159.1,E2 -10159.1} C_VEL
LIN {X 0,Y 417.617,Z 541.873,A -85,B 0,C 180,E1 -10160.8,E2 -10160.8} C_VEL
LIN {X 0,Y 417.318,Z 546.589,A -85,B 0,C 180,E1 -10162.257,E2 -10162.257} C_VEL
LIN {X 0,Y 417.129,Z 551.477,A -85,B 0,C 180,E1 -10164.198,E2 -10164.198} C_VEL
LIN {X 0,Y 416.989,Z 554.874,A -85,B 0,C 180,E1 -10166.134,E2 -10166.134} C_VEL
LIN {X 0,Y 417.027,Z 556.884,A -85,B 0,C 180,E1 -10168.068,E2 -10168.068} C_VEL
LIN {X 0,Y 416.981,Z 557.55,A -85,B 0,C 180,E1 -10170,E2 -10170} C_VEL
LIN {X 0,Y 417.027,Z 556.884,A -85,B 0,C 180,E1 -10171.931,E2 -10171.931} C_VEL
LIN {X 0,Y 416.989,Z 554.874,A -85,B 0,C 180,E1 -10173.866,E2 -10173.866} C_VEL
LIN {X 0,Y 417.145,Z 551.473,A -85,B 0,C 180,E1 -10175.802,E2 -10175.802} C_VEL
LIN {X 0,Y 417.317,Z 546.578,A -85,B 0,C 180,E1 -10177.743,E2 -10177.743} C_VEL
LIN {X 0,Y 417.761,Z 540.046,A -85,B 0,C 180,E1 -10179.685,E2 -10179.685} C_VEL
LIN {X 0,Y 418.33,Z 532.777,A -85,B 0,C 180,E1 -10181.385,E2 -10181.385} C_VEL
LIN {X 0,Y 418.985,Z 524.305,A -85,B 0,C 180,E1 -10182.996,E2 -10182.996} C_VEL
LIN {X 0,Y 419.836,Z 514.324,A -85,B 0,C 180,E1 -10184.542,E2 -10184.542} C_VEL
LIN {X 0,Y 420.78,Z 503.863,A -85,B 0,C 180,E1 -10185.873,E2 -10185.873} C_VEL
LIN {X 0,Y 421.825,Z 492.319,A -85,B 0,C 180,E1 -10187.076,E2 -10187.076} C_VEL
LIN {X 0,Y 422.832,Z 479.51,A -85,B 0,C 180,E1 -10188.159,E2 -10188.159} C_VEL
LIN {X 0,Y 423.762,Z 465.824,A -85,B 0,C 180,E1 -10189.068,E2 -10189.068} C_VEL
LIN {X 0,Y 424.142,Z 456.798,A -85,B 0,C 180,E1 -10189.551,E2 -10189.551} C_VEL
LIN {X 0,Y 421.559,Z 443.392,A -85,B 0,C 180,E1 -10190.255,E2 -10190.255} C_VEL
LIN {X 0,Y 418.192,Z 429.439,A -85,B 0,C 180,E1 -10190.834,E2 -10190.834} C_VEL
LIN {X 0,Y 417.532,Z 426.758,A -85,B 0,C 180,E1 -10190.926,E2 -10190.926} C_VEL
LIN {X 0,Y 417.683,Z 421.587,A -85,B 0,C 180,E1 -10193.818,E2 -10193.818} C_VEL
LIN {X 0,Y 417.942,Z 416.062,A -85,B 0,C 180,E1 -10197.002,E2 -10197.002} C_VEL
LIN {X 0,Y 418.264,Z 410.528,A -85,B 0,C 180,E1 -10200.271,E2 -10200.271} C_VEL
LIN {X 0,Y 418.585,Z 405.007,A -85,B 0,C 180,E1 -10203.646,E2 -10203.646} C_VEL
LIN {X 0,Y 418.924,Z 399.5,A -85,B 0,C 180,E1 -10207.153,E2 -10207.153} C_VEL
LIN {X 0,Y 418.911,Z 395.835,A -85,B 0,C 180,E1 -10209.607,E2 -10209.607} C_VEL
LIN {X 0,Y 418.428,Z 391.956,A -85,B 0,C 180,E1 -10212.351,E2 -10212.351} C_VEL
LIN {X 0,Y 418.232,Z 391.016,A -85,B 0,C 180,E1 -10213.229,E2 -10213.229} C_VEL
LIN {X 0,Y 418.21,Z 391.021,A -85,B 0,C 180,E1 -10216.449,E2 -10216.449} C_VEL
LIN {X 0,Y 418.266,Z 391.013,A -85,B 0,C 180,E1 -10219.123,E2 -10219.123} C_VEL
LIN {X 0,Y 418.24,Z 391.013,A -85,B 0,C 180,E1 -10222.165,E2 -10222.165} C_VEL
LIN {X 0,Y 418.267,Z 391.01,A -85,B 0,C 180,E1 -10225.42,E2 -10225.42} C_VEL
LIN {X 0,Y 418.212,Z 391.016,A -85,B 0,C 180,E1 -10228.604,E2 -10228.604} C_VEL
LIN {X 0,Y 418.293,Z 391.006,A -85,B 0,C 180,E1 -10231.937,E2 -10231.937} C_VEL
LIN {X 0,Y 418.291,Z 391.006,A -85,B 0,C 180,E1 -10235.163,E2 -10235.163} C_VEL
LIN {X 0,Y 418.235,Z 391.012,A -85,B 0,C 180,E1 -10238.304,E2 -10238.304} C_VEL
LIN {X 0,Y 418.286,Z 391.005,A -85,B 0,C 180,E1 -10241.383,E2 -10241.383} C_VEL
LIN {X 0,Y 418.313,Z 391.002,A -85,B 0,C 180,E1 -10244.406,E2 -10244.406} C_VEL
LIN {X 0,Y 418.357,Z 390.998,A -85,B 0,C 180,E1 -10247.386,E2 -10247.386} C_VEL
LIN {X 0,Y 418.343,Z 391.002,A -85,B 0,C 180,E1 -10250.329,E2 -10250.329} C_VEL
LIN {X 0,Y 418.515,Z 390.975,A -85,B 0,C 180,E1 -10252.28,E2 -10252.28} C_VEL
LIN {X 0,Y 418.515,Z 390.977,A -85,B 0,C 180,E1 -10254.217,E2 -10254.217} C_VEL
LIN {X 0,Y 418.547,Z 390.974,A -85,B 0,C 180,E1 -10258.076,E2 -10258.076} C_VEL
LIN {X 0,Y 418.675,Z 390.96,A -85,B 0,C 180,E1 -10260,E2 -10260} C_VEL
LIN {X 0,Y 418.503,Z 390.979,A -85,B 0,C 180,E1 -10262.888,E2 -10262.888} C_VEL
LIN {X 0,Y 418.496,Z 390.982,A -85,B 0,C 180,E1 -10266.751,E2 -10266.751} C_VEL
LIN {X 0,Y 418.359,Z 391,A -85,B 0,C 180,E1 -10269.671,E2 -10269.671} C_VEL
LIN {X 0,Y 418.348,Z 390.999,A -85,B 0,C 180,E1 -10273.001,E2 -10273.001} C_VEL
LIN {X 0,Y 418.322,Z 390.999,A -85,B 0,C 180,E1 -10276.739,E2 -10276.739} C_VEL
LIN {X 0,Y 418.273,Z 391.009,A -85,B 0,C 180,E1 -10279.791,E2 -10279.791} C_VEL
LIN {X 0,Y 418.24,Z 391.015,A -85,B 0,C 180,E1 -10282.736,E2 -10282.736} C_VEL
LIN {X 0,Y 418.273,Z 391.011,A -85,B 0,C 180,E1 -10285.904,E2 -10285.904} C_VEL
LIN {X 0,Y 418.266,Z 391.012,A -85,B 0,C 180,E1 -10289.162,E2 -10289.162} C_VEL
LIN {X 0,Y 418.259,Z 391.011,A -85,B 0,C 180,E1 -10292.844,E2 -10292.844} C_VEL
LIN {X 0,Y 418.25,Z 391.011,A -85,B 0,C 180,E1 -10296.239,E2 -10296.239} C_VEL
LIN {X 0,Y 418.254,Z 391.009,A -85,B 0,C 180,E1 -10299.682,E2 -10299.682} C_VEL
LIN {X 0,Y 418.231,Z 391.016,A -85,B 0,C 180,E1 -10302.321,E2 -10302.321} C_VEL
LIN {X 0,Y 418.242,Z 391.014,A -85,B 0,C 180,E1 -10305.109,E2 -10305.109} C_VEL
LIN {X 0,Y 418.244,Z 391.013,A -85,B 0,C 180,E1 -10307.767,E2 -10307.767} C_VEL
LIN {X 0,Y 418.283,Z 391.38,A -85,B 0,C 180,E1 -10309.121,E2 -10309.121} C_VEL
LIN {X 0,Y 418.49,Z 394.492,A -85,B 0,C 180,E1 -10311.584,E2 -10311.584} C_VEL
LIN {X 0,Y 418.481,Z 397.693,A -85,B 0,C 180,E1 -10313.999,E2 -10313.999} C_VEL
LIN {X 0,Y 418.241,Z 402.476,A -85,B 0,C 180,E1 -10317.472,E2 -10317.472} C_VEL
LIN {X 0,Y 418.045,Z 405.654,A -85,B 0,C 180,E1 -10319.712,E2 -10319.712} C_VEL
LIN {X 0,Y 417.852,Z 410.514,A -85,B 0,C 180,E1 -10323.053,E2 -10323.053} C_VEL
LIN {X 0,Y 417.596,Z 415.188,A -85,B 0,C 180,E1 -10326.177,E2 -10326.177} C_VEL
LIN {X 0,Y 417.502,Z 419.735,A -85,B 0,C 180,E1 -10329.129,E2 -10329.129} C_VEL
LIN {X 0,Y 421.312,Z 434.287,A -85,B 0,C 180,E1 -10329.727,E2 -10329.727} C_VEL
LIN {X 0,Y 424.073,Z 446.995,A -85,B 0,C 180,E1 -10330.392,E2 -10330.392} C_VEL
LIN {X 0,Y 424.336,Z 450.832,A -85,B 0,C 180,E1 -10330.593,E2 -10330.593} C_VEL
LIN {X 0,Y 423.554,Z 464.755,A -85,B 0,C 180,E1 -10331.404,E2 -10331.404} C_VEL
LIN {X 0,Y 422.643,Z 477.233,A -85,B 0,C 180,E1 -10332.334,E2 -10332.334} C_VEL
LIN {X 0,Y 421.435,Z 490.118,A -85,B 0,C 180,E1 -10333.531,E2 -10333.531} C_VEL
LIN {X 0,Y 420.544,Z 500.634,A -85,B 0,C 180,E1 -10334.739,E2 -10334.739} C_VEL
LIN {X 0,Y 419.727,Z 509.776,A -85,B 0,C 180,E1 -10335.998,E2 -10335.998} C_VEL
LIN {X 0,Y 419.084,Z 518.335,A -85,B 0,C 180,E1 -10337.408,E2 -10337.408} C_VEL
LIN {X 0,Y 418.255,Z 526.842,A -85,B 0,C 180,E1 -10339.104,E2 -10339.104} C_VEL
LIN {X 0,Y 417.764,Z 533.693,A -85,B 0,C 180,E1 -10340.804,E2 -10340.804} C_VEL
LIN {X 0,Y 417.424,Z 538.423,A -85,B 0,C 180,E1 -10342.259,E2 -10342.259} C_VEL
LIN {X 0,Y 417.305,Z 541.851,A -85,B 0,C 180,E1 -10343.537,E2 -10343.537} C_VEL
LIN {X 0,Y 417.141,Z 545.206,A -85,B 0,C 180,E1 -10345.168,E2 -10345.168} C_VEL
LIN {X 0,Y 417.031,Z 547.916,A -85,B 0,C 180,E1 -10347.102,E2 -10347.102} C_VEL
LIN {X 0,Y 416.991,Z 549.274,A -85,B 0,C 180,E1 -10349.034,E2 -10349.034} C_VEL
LIN {X 0,Y 416.992,Z 549.31,A -85,B 0,C 180,E1 -10350.966,E2 -10350.966} C_VEL
LIN {X 0,Y 417.03,Z 548.02,A -85,B 0,C 180,E1 -10352.898,E2 -10352.898} C_VEL
LIN {X 0,Y 417.069,Z 546.047,A -85,B 0,C 180,E1 -10354.397,E2 -10354.397} C_VEL
LIN {X 0,Y 416.494,Z 544.764,A -85,B 0,C 180,E1 -10355.186,E2 -10355.186} C_VEL
LIN {X 0,Y 413.75,Z 542.311,A -85,B 0,C 180,E1 -10356.459,E2 -10356.459} C_VEL
LIN {X 0,Y 411.442,Z 539.921,A -85,B 0,C 180,E1 -10357.467,E2 -10357.467} C_VEL
LIN {X 0,Y 410.522,Z 537.771,A -85,B 0,C 180,E1 -10358.229,E2 -10358.229} C_VEL
LIN {X 0,Y 410.488,Z 536.976,A -85,B 0,C 180,E1 -10358.482,E2 -10358.482} C_VEL
LIN {X 0,Y 411.008,Z 530.406,A -85,B 0,C 180,E1 -10360.343,E2 -10360.343} C_VEL
LIN {X 0,Y 411.709,Z 522.735,A -85,B 0,C 180,E1 -10362.07,E2 -10362.07} C_VEL
LIN {X 0,Y 412.354,Z 514.771,A -85,B 0,C 180,E1 -10363.547,E2 -10363.547} C_VEL
LIN {X 0,Y 413.275,Z 505.077,A -85,B 0,C 180,E1 -10365.031,E2 -10365.031} C_VEL
LIN {X 0,Y 414.322,Z 494.361,A -85,B 0,C 180,E1 -10366.38,E2 -10366.38} C_VEL
LIN {X 0,Y 415.399,Z 482.487,A -85,B 0,C 180,E1 -10367.603,E2 -10367.603} C_VEL
LIN {X 0,Y 416.37,Z 470.817,A -85,B 0,C 180,E1 -10368.578,E2 -10368.578} C_VEL
LIN {X 0,Y 417.267,Z 457.682,A -85,B 0,C 180,E1 -10369.456,E2 -10369.456} C_VEL
LIN {X 0,Y 417.68,Z 450.414,A -85,B 0,C 180,E1 -10369.852,E2 -10369.852} C_VEL
LIN {X 0,Y 415.058,Z 437.252,A -85,B 0,C 180,E1 -10370.586,E2 -10370.586} C_VEL
LIN {X 0,Y 411.264,Z 423.105,A -85,B 0,C 180,E1 -10371.228,E2 -10371.228} C_VEL
LIN {X 0,Y 410.408,Z 419.717,A -85,B 0,C 180,E1 -10371.373,E2 -10371.373} C_VEL
LIN {X 0,Y 410.651,Z 413.808,A -85,B 0,C 180,E1 -10375.332,E2 -10375.332} C_VEL
LIN {X 0,Y 410.801,Z 410.634,A -85,B 0,C 180,E1 -10377.511,E2 -10377.511} C_VEL
LIN {X 0,Y 411.106,Z 405.285,A -85,B 0,C 180,E1 -10381.266,E2 -10381.266} C_VEL
LIN {X 0,Y 411.303,Z 401.077,A -85,B 0,C 180,E1 -10384.324,E2 -10384.324} C_VEL
LIN {X 0,Y 411.47,Z 397.869,A -85,B 0,C 180,E1 -10386.713,E2 -10386.713} C_VEL
LIN {X 0,Y 411.441,Z 393.955,A -85,B 0,C 180,E1 -10389.766,E2 -10389.766} C_VEL
LIN {X 0,Y 411.234,Z 392.159,A -85,B 0,C 180,E1 -10391.239,E2 -10391.239} C_VEL
LIN {X 0,Y 411.184,Z 391.895,A -85,B 0,C 180,E1 -10393.132,E2 -10393.132} C_VEL
LIN {X 0,Y 411.171,Z 391.896,A -85,B 0,C 180,E1 -10395.881,E2 -10395.881} C_VEL
LIN {X 0,Y 411.166,Z 391.896,A -85,B 0,C 180,E1 -10398.772,E2 -10398.772} C_VEL
LIN {X 0,Y 411.203,Z 391.888,A -85,B 0,C 180,E1 -10402.027,E2 -10402.027} C_VEL
LIN {X 0,Y 411.209,Z 391.889,A -85,B 0,C 180,E1 -10405.667,E2 -10405.667} C_VEL
LIN {X 0,Y 411.192,Z 391.893,A -85,B 0,C 180,E1 -10409.152,E2 -10409.152} C_VEL
LIN {X 0,Y 411.262,Z 391.884,A -85,B 0,C 180,E1 -10412.522,E2 -10412.522} C_VEL
LIN {X 0,Y 411.23,Z 391.885,A -85,B 0,C 180,E1 -10415.785,E2 -10415.785} C_VEL
LIN {X 0,Y 411.199,Z 391.889,A -85,B 0,C 180,E1 -10418.966,E2 -10418.966} C_VEL
LIN {X 0,Y 411.255,Z 391.885,A -85,B 0,C 180,E1 -10422.085,E2 -10422.085} C_VEL
LIN {X 0,Y 411.264,Z 391.881,A -85,B 0,C 180,E1 -10425.147,E2 -10425.147} C_VEL
LIN {X 0,Y 411.287,Z 391.878,A -85,B 0,C 180,E1 -10428.167,E2 -10428.167} C_VEL
LIN {X 0,Y 411.485,Z 391.855,A -85,B 0,C 180,E1 -10432.147,E2 -10432.147} C_VEL
LIN {X 0,Y 411.478,Z 391.854,A -85,B 0,C 180,E1 -10434.118,E2 -10434.118} C_VEL
LIN {X 0,Y 411.514,Z 391.85,A -85,B 0,C 180,E1 -10438.042,E2 -10438.042} C_VEL
LIN {X 0,Y 411.643,Z 391.837,A -85,B 0,C 180,E1 -10440,E2 -10440} C_VEL
LIN {X 0,Y 411.468,Z 391.856,A -85,B 0,C 180,E1 -10442.937,E2 -10442.937} C_VEL
LIN {X 0,Y 411.464,Z 391.857,A -85,B 0,C 180,E1 -10446.867,E2 -10446.867} C_VEL
LIN {X 0,Y 411.307,Z 391.878,A -85,B 0,C 180,E1 -10449.838,E2 -10449.838} C_VEL
LIN {X 0,Y 411.308,Z 391.879,A -85,B 0,C 180,E1 -10453.104,E2 -10453.104} C_VEL
LIN {X 0,Y 411.265,Z 391.879,A -85,B 0,C 180,E1 -10456.869,E2 -10456.869} C_VEL
LIN {X 0,Y 411.233,Z 391.885,A -85,B 0,C 180,E1 -10459.987,E2 -10459.987} C_VEL
LIN {X 0,Y 411.206,Z 391.886,A -85,B 0,C 180,E1 -10463.147,E2 -10463.147} C_VEL
LIN {X 0,Y 411.24,Z 391.883,A -85,B 0,C 180,E1 -10466.381,E2 -10466.381} C_VEL
LIN {X 0,Y 411.203,Z 391.886,A -85,B 0,C 180,E1 -10469.713,E2 -10469.713} C_VEL
LIN {X 0,Y 411.208,Z 391.888,A -85,B 0,C 180,E1 -10473.156,E2 -10473.156} C_VEL
LIN {X 0,Y 411.198,Z 391.891,A -85,B 0,C 180,E1 -10476.553,E2 -10476.553} C_VEL
LIN {X 0,Y 411.23,Z 391.888,A -85,B 0,C 180,E1 -10479.73,E2 -10479.73} C_VEL
LIN {X 0,Y 411.179,Z 391.894,A -85,B 0,C 180,E1 -10483.133,E2 -10483.133} C_VEL
LIN {X 0,Y 411.202,Z 391.913,A -85,B 0,C 180,E1 -10486.702,E2 -10486.702} C_VEL
LIN {X 0,Y 411.787,Z 395.816,A -85,B 0,C 180,E1 -10489.567,E2 -10489.567} C_VEL
LIN {X 0,Y 411.931,Z 399.481,A -85,B 0,C 180,E1 -10492.106,E2 -10492.106} C_VEL
LIN {X 0,Y 411.669,Z 403.922,A -85,B 0,C 180,E1 -10495.03,E2 -10495.03} C_VEL
LIN {X 0,Y 411.38,Z 408.648,A -85,B 0,C 180,E1 -10498.021,E2 -10498.021} C_VEL
LIN {X 0,Y 411.037,Z 414.171,A -85,B 0,C 180,E1 -10501.396,E2 -10501.396} C_VEL
LIN {X 0,Y 410.727,Z 419.698,A -85,B 0,C 180,E1 -10504.673,E2 -10504.673} C_VEL
LIN {X 0,Y 410.497,Z 426.147,A -85,B 0,C 180,E1 -10508.402,E2 -10508.402} C_VEL
LIN {X 0,Y 410.482,Z 426.65,A -85,B 0,C 180,E1 -10508.688,E2 -10508.688} C_VEL
LIN {X 0,Y 414.242,Z 441.879,A -85,B 0,C 180,E1 -10509.314,E2 -10509.314} C_VEL
LIN {X 0,Y 416.832,Z 454.697,A -85,B 0,C 180,E1 -10509.986,E2 -10509.986} C_VEL
LIN {X 0,Y 417.442,Z 459.012,A -85,B 0,C 180,E1 -10510.235,E2 -10510.235} C_VEL
LIN {X 0,Y 416.679,Z 472.144,A -85,B 0,C 180,E1 -10511.011,E2 -10511.011} C_VEL
LIN {X 0,Y 415.702,Z 484.11,A -85,B 0,C 180,E1 -10511.901,E2 -10511.901} C_VEL
LIN {X 0,Y 414.658,Z 496.005,A -85,B 0,C 180,E1 -10513,E2 -10513} C_VEL
LIN {X 0,Y 413.684,Z 506.869,A -85,B 0,C 180,E1 -10514.227,E2 -10514.227} C_VEL
LIN {X 0,Y 412.62,Z 517.604,A -85,B 0,C 180,E1 -10515.701,E2 -10515.701} C_VEL
LIN {X 0,Y 411.857,Z 526.467,A -85,B 0,C 180,E1 -10517.183,E2 -10517.183} C_VEL
LIN {X 0,Y 411.092,Z 534.96,A -85,B 0,C 180,E1 -10518.911,E2 -10518.911} C_VEL
LIN {X 0,Y 410.578,Z 541.805,A -85,B 0,C 180,E1 -10520.641,E2 -10520.641} C_VEL
LIN {X 0,Y 410.259,Z 546.521,A -85,B 0,C 180,E1 -10522.123,E2 -10522.123} C_VEL
LIN {X 0,Y 410.053,Z 551.409,A -85,B 0,C 180,E1 -10524.097,E2 -10524.097} C_VEL
LIN {X 0,Y 409.909,Z 554.806,A -85,B 0,C 180,E1 -10526.067,E2 -10526.067} C_VEL
LIN {X 0,Y 409.923,Z 556.816,A -85,B 0,C 180,E1 -10528.035,E2 -10528.035} C_VEL
LIN {X 0,Y 409.904,Z 557.481,A -85,B 0,C 180,E1 -10530,E2 -10530} C_VEL
LIN {X 0,Y 409.923,Z 556.815,A -85,B 0,C 180,E1 -10531.965,E2 -10531.965} C_VEL
LIN {X 0,Y 409.909,Z 554.804,A -85,B 0,C 180,E1 -10533.932,E2 -10533.932} C_VEL
LIN {X 0,Y 410.069,Z 551.404,A -85,B 0,C 180,E1 -10535.902,E2 -10535.902} C_VEL
LIN {X 0,Y 410.259,Z 546.508,A -85,B 0,C 180,E1 -10537.877,E2 -10537.877} C_VEL
LIN {X 0,Y 410.739,Z 539.976,A -85,B 0,C 180,E1 -10539.852,E2 -10539.852} C_VEL
LIN {X 0,Y 411.339,Z 532.707,A -85,B 0,C 180,E1 -10541.581,E2 -10541.581} C_VEL
LIN {X 0,Y 411.976,Z 524.755,A -85,B 0,C 180,E1 -10543.125,E2 -10543.125} C_VEL
LIN {X 0,Y 412.778,Z 515.945,A -85,B 0,C 180,E1 -10544.545,E2 -10544.545} C_VEL
LIN {X 0,Y 413.826,Z 504.858,A -85,B 0,C 180,E1 -10546.02,E2 -10546.02} C_VEL
LIN {X 0,Y 414.906,Z 493.539,A -85,B 0,C 180,E1 -10547.243,E2 -10547.243} C_VEL
LIN {X 0,Y 415.947,Z 481.02,A -85,B 0,C 180,E1 -10548.342,E2 -10548.342} C_VEL
LIN {X 0,Y 416.941,Z 467.57,A -85,B 0,C 180,E1 -10549.276,E2 -10549.276} C_VEL
LIN {X 0,Y 417.408,Z 458.921,A -85,B 0,C 180,E1 -10549.766,E2 -10549.766} C_VEL
LIN {X 0,Y 415.317,Z 446.617,A -85,B 0,C 180,E1 -10550.447,E2 -10550.447} C_VEL
LIN {X 0,Y 411.912,Z 432.393,A -85,B 0,C 180,E1 -10551.097,E2 -10551.097} C_VEL
LIN {X 0,Y 410.489,Z 426.689,A -85,B 0,C 180,E1 -10551.302,E2 -10551.302} C_VEL
LIN {X 0,Y 410.708,Z 420.39,A -85,B 0,C 180,E1 -10554.915,E2 -10554.915} C_VEL
